(* IEC 61131-3 sources: Industry-PLC-LLM/data/PLCBEAD_repo/PLCBEAD_PLCEmbed-main/PLC-BEAD/Source/GEB/sample_project/oscat/Network (part 2) *)

(* ---- NET_VAR_BOOL8.ST ---- *)
TYPE

	oscat_NW_BUF_LONG  : ARRAY [0..4095] OF BYTE;

	oscat_NETWORK_BUFFER :
	STRUCT
		SIZE   : UINT;
		BUFFER : oscat_NW_BUF_LONG;
	END_STRUCT;

END_TYPE

TYPE oscat_NET_VAR_DATA :
	STRUCT
		CYCLE : UDINT;
		STATE : BYTE;
		INDEX : INT;
		ID_MAX : USINT;
		ERROR_ID : BYTE;
		BUF_SIZE : UINT;
		S_BUF : oscat_NETWORK_BUFFER;
		R_BUF : oscat_NETWORK_BUFFER;
	END_STRUCT;
END_TYPE

FUNCTION BIT_OF_DWORD : BOOL
  VAR_INPUT
    IN : DWORD;
    N : INT;
  END_VAR

  BIT_OF_DWORD := (SHR(IN,N) AND 16#00000001) > 0;
END_FUNCTION

FUNCTION_BLOCK BYTE_TO_BITS_Block
	VAR_INPUT
		IN :	BYTE;
	END_VAR

	VAR_OUTPUT
		B0 :	BOOL;
		B1 :	BOOL;
		B2 :	BOOL;
		B3 :	BOOL;
		B4 :	BOOL;
		B5 :	BOOL;
		B6 :	BOOL;
		B7 :	BOOL;
	END_VAR

	B0 := BIT_OF_DWORD(BYTE_TO_DWORD(IN),0); (* IN.X0 *)
	B1 := BIT_OF_DWORD(BYTE_TO_DWORD(IN),1); (* IN.X1 *)
	B2 := BIT_OF_DWORD(BYTE_TO_DWORD(IN),2); (* IN.X2 *)
	B3 := BIT_OF_DWORD(BYTE_TO_DWORD(IN),3); (* IN.X3 *)
	B4 := BIT_OF_DWORD(BYTE_TO_DWORD(IN),4); (* IN.X4 *)
	B5 := BIT_OF_DWORD(BYTE_TO_DWORD(IN),5); (* IN.X5 *)
	B6 := BIT_OF_DWORD(BYTE_TO_DWORD(IN),6); (* IN.X6 *)
	B7 := BIT_OF_DWORD(BYTE_TO_DWORD(IN),7); (* IN.X7 *)
END_FUNCTION_BLOCK

FUNCTION BYTE_OF_BIT:BYTE
	VAR_INPUT
		B0 :	BOOL;
		B1 :	BOOL;
		B2 :	BOOL;
		B3 :	BOOL;
		B4 :	BOOL;
		B5 :	BOOL;
		B6 :	BOOL;
		B7 :	BOOL;
	END_VAR
	Byte_of_bit := SHL(SHL(SHL(SHL(SHL(SHL(SHL(BOOL_TO_BYTE(B7),1) OR BOOL_TO_BYTE(B6),1)
	OR BOOL_TO_BYTE(B5),1) OR BOOL_TO_BYTE(B4),1) OR BOOL_TO_BYTE(B3),1) OR BOOL_TO_BYTE(B2),1)
	OR BOOL_TO_BYTE(B1),1) OR BOOL_TO_BYTE(B0);
END_FUNCTION

FUNCTION_BLOCK NET_VAR_BOOL8_Block

	VAR_INPUT
		IN1 :	BOOL;
		IN2 :	BOOL;
		IN3 :	BOOL;
		IN4 :	BOOL;
		IN5 :	BOOL;
		IN6 :	BOOL;
		IN7 :	BOOL;
		IN8 :	BOOL;
	END_VAR

	VAR_OUTPUT
		OUT1 :	BOOL;
		OUT2 :	BOOL;
		OUT3 :	BOOL;
		OUT4 :	BOOL;
		OUT5 :	BOOL;
		OUT6 :	BOOL;
		OUT7 :	BOOL;
		OUT8 :	BOOL;
		ID :	BYTE;
	END_VAR

	VAR_IN_OUT
		X :	oscat_NET_VAR_DATA;
	END_VAR

	VAR
		init :	BOOL;
		index :	INT;
		indeX2 :	INT;
		_BYTE_TO_BITS :	BYTE_TO_BITS_Block;
	END_VAR

	IF NOT init THEN
		init := TRUE;
		X.ID_MAX := X.ID_MAX + USINT#1;
		ID := USINT_TO_BYTE(X.ID_MAX);
	END_IF;

	IF X.STATE > BYTE#0 AND X.ERROR_ID = BYTE#0 THEN
		index := X.index;
		IF INT_TO_UINT(index + 3) > X.BUF_SIZE THEN
			X.ERROR_ID := ID;
		ELSE
			IF X.STATE = BYTE#1 THEN
				X.S_BUF.BUFFER[index] := ID;
				index := index + 1;
				X.S_BUF.BUFFER[index] := BYTE#4;
				index := index + 1;
				X.S_BUF.BUFFER[index] := BYTE_OF_BIT(IN1,IN2,IN3,IN4,IN5,IN6,IN7,IN8);
				index := index + 1;

			ELSIF X.STATE = BYTE#2 THEN
				indeX2 := index + 1;
				IF X.R_BUF.BUFFER[index] <> ID OR X.R_BUF.BUFFER[indeX2] <> BYTE#4 THEN
					X.ERROR_ID := ID;
				ELSE
					index := index + 2;
					_BYTE_TO_BITS(IN:=X.R_BUF.BUFFER[index]);
					OUT1 := _BYTE_TO_BITS.B0;
					OUT2 := _BYTE_TO_BITS.B1;
					OUT3 := _BYTE_TO_BITS.B2;
					OUT4 := _BYTE_TO_BITS.B3;
					OUT5 := _BYTE_TO_BITS.B4;
					OUT6 := _BYTE_TO_BITS.B5;
					OUT7 := _BYTE_TO_BITS.B6;
					OUT8 := _BYTE_TO_BITS.B7;
					index := index + 1;
				END_IF;
			END_IF;
			X.index := index;
		END_IF;
	END_IF;

END_FUNCTION_BLOCK

PROGRAM program0
	VAR
		IN1 :	BOOL;
		IN2 :	BOOL;
		IN3 :	BOOL;
		IN4 :	BOOL;
		IN5 :	BOOL;
		IN6 :	BOOL;
		IN7 :	BOOL;
		IN8 :	BOOL;
		OUT1 :	BOOL;
		OUT2 :	BOOL;
		OUT3 :	BOOL;
		OUT4 :	BOOL;
		OUT5 :	BOOL;
		OUT6 :	BOOL;
		OUT7 :	BOOL;
		OUT8 :	BOOL;
		ID :	BYTE;
		X :	oscat_NET_VAR_DATA;

		func_block : NET_VAR_BOOL8_Block;
	END_VAR
	func_block.IN1 := IN1;
	func_block.IN2 := IN2;
	func_block.IN3 := IN3;
	func_block.IN4 := IN4;
	func_block.IN5 := IN5;
	func_block.IN6 := IN6;
	func_block.IN7 := IN7;
	func_block.IN8 := IN8;
	func_block.X := X;

	func_block();
  	OUT1  := func_block.OUT1;
	OUT2  := func_block.OUT2;
	OUT3  := func_block.OUT3;
	OUT4  := func_block.OUT4;
	OUT5  := func_block.OUT5;
	OUT6  := func_block.OUT6;
	OUT7  := func_block.OUT7;
	OUT8  := func_block.OUT8;
	ID  := func_block.ID;
	X  := func_block.X;
END_PROGRAM

CONFIGURATION Config0
	RESOURCE ReS0 ON PLC
		TASK task0(INTERVAL := T#20ms,PRIORITY := 0);
		PROGRAM instance0 WITH task0 : program0;
	END_RESOURCE
END_CONFIGURATION

(* ---- NET_VAR_BUFFER.ST ---- *)
TYPE
	oscat_aB1_64 : ARRAY[1..64] OF BYTE;
END_TYPE

TYPE

	oscat_NW_BUF_LONG  : ARRAY [0..4095] OF BYTE;

	oscat_NETWORK_BUFFER :
	STRUCT
		SIZE   : UINT;
		BUFFER : oscat_NW_BUF_LONG;
	END_STRUCT;

END_TYPE

TYPE oscat_NET_VAR_DATA :
	STRUCT
		CYCLE : UDINT;
		STATE : BYTE;
		INDEX : INT;
		ID_MAX : USINT;
		ERROR_ID : BYTE;
		BUF_SIZE : UINT;
		S_BUF : oscat_NETWORK_BUFFER;
		R_BUF : oscat_NETWORK_BUFFER;
	END_STRUCT;
END_TYPE

FUNCTION_BLOCK NET_VAR_BUFFER_Block

	VAR_OUTPUT
		ID :	BYTE;
	END_VAR

	VAR_IN_OUT
		BUF_IN :	oscat_aB1_64;
		BUF_OUT :	oscat_aB1_64;
		X :	oscat_NET_VAR_DATA;
	END_VAR

	VAR
		SIZE :	INT;
		init :	BOOL;
		index :	INT;
		indeX2 :	INT;
	END_VAR

	IF NOT init THEN
		init := TRUE;
		X.ID_MAX := X.ID_MAX + USINT#1;
		ID := USINT_TO_BYTE(X.ID_MAX);
	END_IF;

	IF X.STATE > BYTE#0 AND X.ERROR_ID = BYTE#0 THEN
		index := X.index;
		IF X.STATE = BYTE#1 THEN
			SIZE := 64;
			IF INT_TO_UINT(index + 3 + SIZE) > X.BUF_SIZE THEN
				X.ERROR_ID := ID;
			ELSE
				X.S_BUF.BUFFER[index] := ID;
				index := index + 1;
				X.S_BUF.BUFFER[index] := BYTE#20;
				index := index + 1;
				X.S_BUF.BUFFER[index] := INT_TO_BYTE(SIZE);
				index := index + 1;
				FOR indeX2 := 1 TO SIZE DO
					X.S_BUF.BUFFER[index] := BUF_IN[indeX2];
					index := index + 1;
				END_FOR;
			END_IF;
		ELSIF X.STATE = BYTE#2 THEN
			indeX2 := index + 1;
			IF X.R_BUF.BUFFER[index] <> ID OR X.R_BUF.BUFFER[indeX2] <> BYTE#20 THEN
				X.ERROR_ID := ID;
			ELSE
				index := index + 2;
				SIZE := BYTE_TO_INT(X.R_BUF.BUFFER[index]);
				index := index + 1;
				FOR indeX2 := 1 TO SIZE DO
					BUF_OUT[indeX2] := X.R_BUF.BUFFER[index];
					index := index + 1;
				END_FOR;
			END_IF;
		END_IF;
		X.index := index;
	END_IF;

END_FUNCTION_BLOCK

PROGRAM program0
	VAR
		BUF_IN :	oscat_aB1_64;
		BUF_OUT :	oscat_aB1_64;
		X :	oscat_NET_VAR_DATA;
		ID :	BYTE;

		func_block : NET_VAR_BUFFER_Block;
	END_VAR
	func_block.BUF_IN := BUF_IN;
	func_block.BUF_OUT := BUF_OUT;
	func_block.X := X;

	func_block();
  	BUF_IN  := func_block.BUF_IN;
	BUF_OUT  := func_block.BUF_OUT;
	X  := func_block.X;
	ID  := func_block.ID;

END_PROGRAM

CONFIGURATION Config0
	RESOURCE ReS0 ON PLC
		TASK task0(INTERVAL := T#20ms,PRIORITY := 0);
		PROGRAM instance0 WITH task0 : program0;
	END_RESOURCE
END_CONFIGURATION

(* ---- NET_VAR_DWORD8.ST ---- *)
TYPE
	oscat_nv_dw : ARRAY[1..8] OF DWORD;
END_TYPE

TYPE

	oscat_NW_BUF_LONG  : ARRAY [0..4095] OF BYTE;

	oscat_NETWORK_BUFFER :
	STRUCT
		SIZE   : UINT;
		BUFFER : oscat_NW_BUF_LONG;
	END_STRUCT;

END_TYPE

TYPE oscat_NET_VAR_DATA :
	STRUCT
		CYCLE : UDINT;
		STATE : BYTE;
		INDEX : INT;
		ID_MAX : USINT;
		ERROR_ID : BYTE;
		BUF_SIZE : UINT;
		S_BUF : oscat_NETWORK_BUFFER;
		R_BUF : oscat_NETWORK_BUFFER;
	END_STRUCT;
END_TYPE

FUNCTION_BLOCK NET_VAR_DWORD8_Block

	VAR_INPUT
		IN1 :	DWORD;
		IN2 :	DWORD;
		IN3 :	DWORD;
		IN4 :	DWORD;
		IN5 :	DWORD;
		IN6 :	DWORD;
		IN7 :	DWORD;
		IN8 :	DWORD;
	END_VAR

	VAR_OUTPUT
		OUT1 :	DWORD;
		OUT2 :	DWORD;
		OUT3 :	DWORD;
		OUT4 :	DWORD;
		OUT5 :	DWORD;
		OUT6 :	DWORD;
		OUT7 :	DWORD;
		OUT8 :	DWORD;
		ID :	BYTE;
	END_VAR

	VAR_IN_OUT
		X :	oscat_NET_VAR_DATA;
	END_VAR

	VAR
		init :	BOOL;
		i :	INT;
		i2 :	INT;
		index :	INT;
		indeX2 :	INT;
		ra :	oscat_nv_dw;
	END_VAR

	IF NOT init THEN
		init := TRUE;
		X.ID_MAX := X.ID_MAX + USINT#1;
		ID := USINT_TO_BYTE(X.ID_MAX);
	END_IF;

	IF X.STATE > BYTE#0 AND X.ERROR_ID = BYTE#0 THEN
		index := X.index;
		IF INT_TO_UINT(index + 34) > X.BUF_SIZE THEN
			X.ERROR_ID := ID;
		ELSE
			IF X.STATE = BYTE#1 THEN
				ra[1] := IN1;
				ra[2] := IN2;
				ra[3] := IN3;
				ra[4] := IN4;
				ra[5] := IN5;
				ra[6] := IN6;
				ra[7] := IN7;
				ra[8] := IN8;
				X.S_BUF.BUFFER[index] := ID;
				index := index + 1;
				X.S_BUF.BUFFER[index] := BYTE#13;
				index := index + 1;
				FOR i2 := 1 TO 8 DO
					FOR i := 1 TO 4 DO
						X.S_BUF.BUFFER[index] := DWORD_TO_BYTE(ra[i2]);
						ra[i2] := ROR(ra[i2],8);
						index := index + 1;
					END_FOR;
				END_FOR;

			ELSIF X.STATE = BYTE#2 THEN
				indeX2 := index + 1;
				IF X.R_BUF.BUFFER[index] <> ID OR X.R_BUF.BUFFER[indeX2] <> BYTE#13 THEN
					X.ERROR_ID := ID;
				ELSE
					index := index + 2;
					FOR i2 := 1 TO 8 DO
						ra[i2] := DWORD#0;
						FOR i := 1 TO 4 DO
							ra[i2] := ra[i2] OR BYTE_TO_DWORD(X.R_BUF.BUFFER[index]);
							ra[i2] := ROR(ra[i2],8);
							index := index + 1;
						END_FOR;
					END_FOR;
					OUT1 := ra[1];
					OUT2 := ra[2];
					OUT3 := ra[3];
					OUT4 := ra[4];
					OUT5 := ra[5];
					OUT6 := ra[6];
					OUT7 := ra[7];
					OUT8 := ra[8];
				END_IF;
			END_IF;
			X.index := index;
		END_IF;
	END_IF;

END_FUNCTION_BLOCK

PROGRAM program0
	VAR
		IN1 :	DWORD;
		IN2 :	DWORD;
		IN3 :	DWORD;
		IN4 :	DWORD;
		IN5 :	DWORD;
		IN6 :	DWORD;
		IN7 :	DWORD;
		IN8 :	DWORD;
		OUT1 :	DWORD;
		OUT2 :	DWORD;
		OUT3 :	DWORD;
		OUT4 :	DWORD;
		OUT5 :	DWORD;
		OUT6 :	DWORD;
		OUT7 :	DWORD;
		OUT8 :	DWORD;
		ID :	BYTE;
		X :	oscat_NET_VAR_DATA;

		func_block : NET_VAR_DWORD8_Block;
	END_VAR
	func_block.IN1 := IN1;
	func_block.IN2 := IN2;
	func_block.IN3 := IN3;
	func_block.IN4 := IN4;
	func_block.IN5 := IN5;
	func_block.IN6 := IN6;
	func_block.IN7 := IN7;
	func_block.IN8 := IN8;
	func_block.X := X;

	func_block();
  	OUT1  := func_block.OUT1;
	OUT2  := func_block.OUT2;
	OUT3  := func_block.OUT3;
	OUT4  := func_block.OUT4;
	OUT5  := func_block.OUT5;
	OUT6  := func_block.OUT6;
	OUT7  := func_block.OUT7;
	OUT8  := func_block.OUT8;
	ID  := func_block.ID;
	X  := func_block.X;
END_PROGRAM

CONFIGURATION Config0
	RESOURCE ReS0 ON PLC
		TASK task0(INTERVAL := T#20ms,PRIORITY := 0);
		PROGRAM instance0 WITH task0 : program0;
	END_RESOURCE
END_CONFIGURATION

(* ---- SHA1_STREAM.ST ---- *)
TYPE
  oscat_aB0_19	: ARRAY [0..19]	OF BYTE;
  oscat_aB0_63	: ARRAY [0..63]	OF BYTE;
  oscat_aDW0_4	: ARRAY [0..4] 	OF DWORD;
  oscat_sDW0_79	: ARRAY [0..79] OF DWORD;

END_TYPE

FUNCTION DWORD_OF_BYTE:DWORD
	VAR_INPUT
		B3 :	BYTE;
		B2 :	BYTE;
		B1 :	BYTE;
		B0 :	BYTE;
	END_VAR

	DWORD_OF_BYTE := SHL(SHL(SHL(BYTE_TO_DWORD(B3),8) OR BYTE_TO_DWORD(B2),8) OR BYTE_TO_DWORD(B1),8) OR BYTE_TO_DWORD(B0);

END_FUNCTION

FUNCTION_BLOCK SHA1_STREAM_Block

	VAR_IN_OUT
		MODE :	INT;
		BUF :	oscat_aB0_63;
		SHA1 :	oscat_aB0_19;
		SIZE :	UDINT;
	END_VAR

	VAR_OUTPUT
		POS :	UDINT;
	END_VAR

	VAR
		hash :	oscat_aDW0_4;
		end :	UDINT;
		block :	UDINT;
		pad_1 :	BOOL;
		w :	oscat_sDW0_79;
		n :	INT;
		n1 :	INT;
		n2 :	INT;
		n3 :	INT;
		n4 :	INT;
		a :	DWORD;
		b :	DWORD;
		c :	DWORD;
		d :	DWORD;
		e :	DWORD;
		f :	DWORD;
		k :	DWORD;
		x :	DWORD;
	END_VAR

	CASE MODE OF

	1:
		hash[0] := DWORD#16#67452301;
		hash[1] := DWORD#16#EFCDAB89;
		hash[2] := DWORD#16#98BADCFE;
		hash[3] := DWORD#16#10325476;
		hash[4] := DWORD#16#C3D2E1F0;

		FOR n := 16 TO 79 DO
			w[n] := DWORD#0;
		END_FOR;

		block := DWORD_TO_UDINT(SHR(UDINT_TO_DWORD(SIZE),6)) + BOOL_TO_UDINT((UDINT_TO_BYTE(SIZE) AND BYTE#16#3F) > BYTE#55);

		pad_1 := FALSE;
		POS := UDINT#0;
		End := SIZE;
		SIZE := MIN(UDINT#64,End);
		MODE := 2;

	2:	FOR n := UDINT_TO_INT(SIZE) TO 63 DO
			BUF[n] := BYTE#0;
		END_FOR;

		IF SIZE < UDINT#64 AND NOT pad_1 THEN
			BUF[SIZE] := BYTE#2#1000_0000;
			pad_1 := TRUE;
		END_IF;

		POS := POS + SIZE;
		SIZE := MIN(UDINT#64,End - POS);

		n := 0;
		FOR n4 := 0 TO 15 DO
			n1 := n + 1;
			n2 := n + 2;
			n3 := n + 3;
			w[n4] := DWORD_OF_BYTE(BUF[n],BUF[n1],BUF[n2],BUF[n3]);
			n := n + 4;
		END_FOR;

		IF block = UDINT#0 THEN
			w[15] := SHL(UDINT_TO_DWORD(End),3);
			MODE := 3;
		ELSE
			block := block - UDINT#1;
		END_IF;

		FOR n := 16 TO 79 DO
			n1 := n - 3;
			n2 := n - 8;
			n3 := n - 14;
			n4 := n - 16;
			w[n] := ROL(w[n1] XOR w[n2] XOR w[n3] XOR w[n4],1);
		END_FOR;

		a := hash[0];
		b := hash[1];
		c := hash[2];
		d := hash[3];
		e := hash[4];

		FOR n := 0 TO 79 DO
			IF n <= 19 THEN
				f := (b AND c) OR (NOT(b) AND d);
				k := DWORD#16#5A827999;
			ELSIF n <= 39 THEN
				f := b XOR c XOR d;
				k := DWORD#16#6ED9EBA1;
			ELSIF n <= 59 THEN
				f := (b AND c) OR (b AND d) OR (c AND d);
				k := DWORD#16#8F1BBCDC;
			ELSE
				f := b XOR c XOR d;
				k := DWORD#16#CA62C1D6;
			END_IF;

			x := UDINT_TO_DWORD(DWORD_TO_UDINT(ROL(a,5)) + DWORD_TO_UDINT(f) + DWORD_TO_UDINT(e) + DWORD_TO_UDINT(k) + DWORD_TO_UDINT(w[n]));
			e := d;
			d := c;
			c := ROL(b,30);
			b := a;
			a := x;
		END_FOR;

		hash[0] := UDINT_TO_DWORD(DWORD_TO_UDINT(hash[0]) + DWORD_TO_UDINT(a));
		hash[1] := UDINT_TO_DWORD(DWORD_TO_UDINT(hash[1]) + DWORD_TO_UDINT(b));
		hash[2] := UDINT_TO_DWORD(DWORD_TO_UDINT(hash[2]) + DWORD_TO_UDINT(c));
		hash[3] := UDINT_TO_DWORD(DWORD_TO_UDINT(hash[3]) + DWORD_TO_UDINT(d));
		hash[4] := UDINT_TO_DWORD(DWORD_TO_UDINT(hash[4]) + DWORD_TO_UDINT(e));

	END_CASE;

	IF MODE = 3 THEN
		n2 := 0;
		FOR n := 0 TO 4 DO
			FOR n1 := 0 TO 3 DO
				hash[n] := ROL(hash[n],8);
				SHA1[n2] := DWORD_TO_BYTE(hash[n]);
				n2 := n2 + 1;
			END_FOR;
		END_FOR;
	END_IF;

END_FUNCTION_BLOCK

PROGRAM program0
	VAR
		MODE :	INT;
		BUF :	oscat_aB0_63;
		SHA1 :	oscat_aB0_19;
		SIZE :	UDINT;
		POS :	UDINT;

		func_block : SHA1_STREAM_Block;
	END_VAR
	func_block.MODE := MODE;
	func_block.BUF := BUF;
	func_block.SHA1 := SHA1;
	func_block.SIZE := SIZE;

	func_block();
  	MODE  := func_block.MODE;
	BUF  := func_block.BUF;
	SHA1  := func_block.SHA1;
	SIZE  := func_block.SIZE;
	POS  := func_block.POS;
END_PROGRAM

CONFIGURATION Config0
	RESOURCE ReS0 ON PLC
		TASK task0(INTERVAL := T#20ms,PRIORITY := 0);
		PROGRAM instance0 WITH task0 : program0;
	END_RESOURCE
END_CONFIGURATION

(* ---- SNTP_CLIENT.ST ---- *)
TYPE
  oscat_IP_FIFO128_DATA  : ARRAY [1..128] OF BYTE;
  oscat_Mailbox  : ARRAY [1..16] OF BYTE;

  oscat_IP_FIFO_DATA :
  STRUCT
    X       : oscat_IP_FIFO128_DATA; (* IP_ID FIFO Speicher          *)
    Y       : oscat_IP_FIFO128_DATA; (* IP_ID Z�hler                 *)
    ID      : BYTE;                  (* h�chste vergabene id         *)
    MAX_ID  : BYTE;                  (* maximal Anmeldungen pro ID   *)
      INIT    : BOOL;                  (* Initialisierung durchgef�hrt *)
    EMPTY   : BOOL;                  (* FIFO leer                    *)
    FULL    : BOOL;                  (* FIFO voll                    *)
    TOP     : INT;                   (* maximale anzahl IN FIFO      *)
    NW      : INT;                   (* Schreibzeiger                *)
    NR      : INT;                   (* Lesezeiger                   *)
  END_STRUCT;

  oscat_IP_C:
  STRUCT
    C_MODE:			BYTE;          		(*W Mode: TCP/UCP AKTIV/PASSIV                               *)
    C_PORT:         WORD;          		(*W Portnummer                                               *)
    C_IP:           DWORD;         		(*W IP-ADRESSe gepackt wwxxyyzz = www.xxx.yyy.zzz            *)
    C_STATE:        BYTE;          		(*R VerbindungsSTATUS ON/OFF + Flanke ON/OFF                 *)
    C_ENABLE:       BOOL;          		(*W Freigabe f�r Connect                                     *)
    R_OBSERVE:      BOOL;          		(*W Empfang ueberwachen                                      *)
    TIME_RESET:     BOOL;          		(*W Alle Timer ruecksetzen                                   *)
    ERROR:          DWORD;         		(*R vvwwxxyy (vv = CON_ERROR, ww = SEN_ERROR, xx = REC_ERROR *)
    FIFO:           oscat_IP_FIFO_DATA; (*I IP FIFO Struktur                                         *)
    MAILBOX:		oscat_Mailbox;		(*I Mailbox: Datenbereich f�r Bausteindatenaustausch         *)
  END_STRUCT;
END_TYPE

TYPE

  oscat_NW_BUF_LONG  : ARRAY [0..4095] OF BYTE;

  oscat_NETWORK_BUFFER :
  STRUCT
    SIZE   : UINT;
    BUFFER : oscat_NW_BUF_LONG;
  END_STRUCT;

END_TYPE

FUNCTION _BYTE_TO_INT:INT
	VAR_INPUT
		IN :	BYTE;
	END_VAR

	_BYTE_TO_INT := USINT_TO_INT(BYTE_TO_USINT(IN));
END_FUNCTION

FUNCTION_BLOCK IP_FIFO_Block

  VAR_IN_OUT
    FIFO :	oscat_IP_FIFO_DATA;
    ID :	BYTE;
    STATE :	BYTE;
  END_VAR

  VAR
    tmp :	INT;
  END_VAR

  IF NOT FIFO.INIT THEN
    FIFO.INIT		:= TRUE;
    FIFO.NW		:= 1;
    FIFO.NR		:= 1;
    FIFO.EMPTY	:= TRUE;
    FIFO.FULL		:= FALSE;
    FIFO.TOP		:= 128;
    FIFO.MAX_ID	:= BYTE#1;
  END_IF;

  IF ID = BYTE#00 THEN
    IF FIFO.ID < INT_TO_BYTE(FIFO.TOP) THEN
      ID := USINT_TO_BYTE(BYTE_TO_USINT(FIFO.ID) + USINT#1);
      FIFO.ID := ID ;

    ELSIF STATE < BYTE#200 THEN
      STATE := BYTE#255;
    RETURN;
    END_IF;
  END_IF;

  IF STATE = BYTE#1 AND NOT FIFO.FULL THEN
    tmp := _BYTE_TO_INT(ID);
    IF FIFO.Y[tmp] < FIFO.MAX_ID THEN
      FIFO.Y[tmp] := USINT_TO_BYTE(BYTE_TO_USINT(FIFO.Y[tmp]) + USINT#1);
      tmp := FIFO.NW;
      FIFO.X[tmp] := ID;
      IF FIFO.NW = FIFO.TOP THEN FIFO.NW := 1; ELSE FIFO.NW := FIFO.NW + 1; END_IF;
      FIFO.FULL := FIFO.NW = FIFO.NR;
    FIFO.EMPTY := FALSE;
      STATE := BYTE#2;
    END_IF;
  END_IF;

  IF STATE = BYTE#2 AND NOT FIFO.EMPTY THEN
    tmp := FIFO.NR;
    IF ID = FIFO.X[tmp] THEN
      STATE := BYTE#3;
    END_IF;
  END_IF;

  IF STATE = BYTE#4 AND NOT FIFO.EMPTY THEN

    tmp := FIFO.NR;
    IF ID = FIFO.X[tmp] THEN
      tmp := _BYTE_TO_INT(ID);
      FIFO.Y[tmp] := USINT_TO_BYTE(BYTE_TO_USINT(FIFO.Y[tmp]) - USINT#1);

      IF FIFO.NR = FIFO.TOP THEN FIFO.NR := 1; ELSE FIFO.NR := FIFO.NR + 1; END_IF;
      FIFO.EMPTY := FIFO.NR = FIFO.NW;
    FIFO.FULL := FALSE;
    END_IF;
    STATE := BYTE#5;
  END_IF;

END_FUNCTION_BLOCK

FUNCTION_BLOCK T_PLC_MS_block

	VAR_OUTPUT
		T_PLC_MS :	UDINT;
	END_VAR

	VAR
		PLC_TICKS_PER_SEC :	INT;
		PLC_SYS_TICK_CNT :	DINT;
	END_VAR

	VAR
		debug :	BOOL;(*Debug-Mode ON / OFF*)
		N :	INT;(*Debug-Faktor*)
		Offset :	UDINT;(*Debug-Offset*)
		temp :	DWORD := DWORD#1;(*Debug-Offset*)
		MODE :	BOOL;(*modus*)
		faktor :	UDINT;(*Systemtakt-Faktor*)
		init :	BOOL;
		v_plc_ticks_per_sec :	UDINT;
		base :	UDINT := UDINT#1000;
	END_VAR

	IF init = FALSE THEN
		v_plc_ticks_per_sec := INT_TO_UDINT(PLC_TICKS_PER_SEC);
		IF v_plc_ticks_per_sec = UDINT#1024 THEN
			faktor := UDINT#1;
			MODE := FALSE;
		ELSIF v_plc_ticks_per_sec > UDINT#0 THEN
			IF v_plc_ticks_per_sec <= base THEN
				faktor := base / v_plc_ticks_per_sec;
				MODE := FALSE;
			ELSE
				faktor := v_plc_ticks_per_sec / base;
				MODE := TRUE;
			END_IF;
		ELSE
			faktor := UDINT#1;
		END_IF;
		init := TRUE;
	END_IF;

	IF MODE THEN
		T_PLC_MS := DINT_TO_UDINT(PLC_SYS_TICK_CNT) / faktor;
	ELSE
		T_PLC_MS := DINT_TO_UDINT(PLC_SYS_TICK_CNT) * faktor;
	END_IF;

	IF debug THEN
		T_PLC_MS := (DWORD_TO_UDINT(SHL(UDINT_TO_DWORD(T_PLC_MS),N) OR SHL(temp,N)) - UDINT#1) + Offset;
	END_IF;

END_FUNCTION_BLOCK

FUNCTION DWORD_OF_BYTE:DWORD
	VAR_INPUT
		B3 :	BYTE;
		B2 :	BYTE;
		B1 :	BYTE;
		B0 :	BYTE;
	END_VAR

	DWORD_OF_BYTE := SHL(SHL(SHL(BYTE_TO_DWORD(B3),8) OR BYTE_TO_DWORD(B2),8) OR BYTE_TO_DWORD(B1),8) OR BYTE_TO_DWORD(B0);

END_FUNCTION

FUNCTION _WORD_TO_DINT:DINT
	VAR_INPUT
		IN :	WORD;
	END_VAR
	_WORD_TO_DINT := UINT_TO_DINT(WORD_TO_UINT(IN));
END_FUNCTION

FUNCTION WORD_OF_BYTE:WORD
	VAR_INPUT
		B1 :	BYTE;
		B0 :	BYTE;
	END_VAR
	WORD_OF_BYTE := SHL(BYTE_TO_WORD(B1),8) OR BYTE_TO_WORD(B0);
END_FUNCTION

FUNCTION _INT_TO_UDINT:UDINT
	VAR_INPUT
		IN :	INT;
	END_VAR

	_INT_TO_UDINT := DINT_TO_UDINT(INT_TO_DINT(IN));
END_FUNCTION

FUNCTION_BLOCK SNTP_CLIENT_Block

  VAR_IN_OUT
    IP_C :	oscat_IP_C;
    S_BUF :	oscat_NETWORK_BUFFER;
    R_BUF :	oscat_NETWORK_BUFFER;
  END_VAR

  VAR_INPUT
    IP4 :	DWORD;
    ACTIVATE :	BOOL;
  END_VAR

  VAR_OUTPUT
    ERROR :	DWORD;
    DONE_P :	BOOL;
    UDT :	UDINT;
    XMS :	INT;
  END_VAR

  VAR
    IP_STATE :	BYTE;
    IP_ID :	BYTE;
    IP_FIFO :	IP_FIFO_Block;
    i :	INT;
    last :	UDINT;
    STATE :	INT;
    T_PLC_MS :	T_PLC_MS_block;
    TX :	UDINT;
    ACTIVATE_LAST :	BOOL;
    IP4_STORED :	DWORD;
  END_VAR

  T_PLC_MS();
  TX := T_PLC_MS.T_PLC_MS;

  CASE STATE OF
  00:
    DONE_P := FALSE;
    IF ACTIVATE AND NOT ACTIVATE_LAST THEN
      IP4_STORED := IP4;
      STATE := 10;
      ERROR := DWORD#0;
      IP_STATE := BYTE#1;
    END_IF;

  10:
    IF IP_STATE = BYTE#3 THEN

      S_BUF.BUFFER[00] := BYTE#16#1B;
      FOR i := 1 TO 47 DO
        S_BUF.BUFFER[i] := BYTE#16#00;
      END_FOR;

      last := TX;
      STATE := 30;

      IP_C.C_PORT     := WORD#123;
      IP_C.C_IP       := IP4_STORED;
      IP_C.C_MODE     := BYTE#1;
      IP_C.C_ENABLE   := TRUE;
      IP_C.TIME_RESET := TRUE;
      IP_C.R_OBSERVE  := TRUE;
      S_BUF.SIZE      := UINT#48;
      R_BUF.SIZE      := UINT#0;
    END_IF;

  30:
    IF IP_C.ERROR <> DWORD#00 THEN
      ERROR := IP_C.ERROR;
    S_BUF.SIZE := UINT#0;
    R_BUF.SIZE := UINT#0;
      STATE := 0;
    ELSIF S_BUF.SIZE = UINT#0 AND R_BUF.SIZE >= UINT#48 THEN
      UDT := DWORD_TO_UDINT(DWORD_OF_BYTE(R_BUF.BUFFER[40],R_BUF.BUFFER[41],R_BUF.BUFFER[42],R_BUF.BUFFER[43]))- UDINT#2208988800;

      XMS := DWORD_TO_INT(SHR(DINT_TO_DWORD(_WORD_TO_DINT(WORD_OF_BYTE(R_BUF.BUFFER[44],R_BUF.BUFFER[45])) * DINT#1000),16));
      XMS := XMS + DWORD_TO_INT(SHR(UDINT_TO_DWORD(SUB_TIME(TX, last)),1));

      UDT := UDT + _INT_TO_UDINT(XMS / 1000);
      XMS := XMS MOD 1000;

      STATE := 0;
      DONE_P := TRUE;

    END_IF;

    IF STATE = 0 THEN
      IP_C.R_OBSERVE := FALSE;
      IP_STATE := BYTE#4;
    END_IF;

  END_CASE;

  ACTIVATE_LAST := ACTIVATE;

  IP_FIFO(FIFO:=IP_C.FIFO,STATE:=IP_STATE,ID:=IP_ID);
  IP_C.FIFO:=IP_FIFO.FIFO;
  IP_STATE := IP_FIFO.STATE;
  IP_ID:=IP_FIFO.ID;

END_FUNCTION_BLOCK

PROGRAM program0
	VAR
		IP_C :	oscat_IP_C;
    S_BUF :	oscat_NETWORK_BUFFER;
    R_BUF :	oscat_NETWORK_BUFFER;
    IP4 :	DWORD;
    ACTIVATE :	BOOL;
    ERROR :	DWORD;
    DONE_P :	BOOL;
    UDT :	UDINT;
    XMS :	INT;

		func_block : SNTP_CLIENT_Block;
	END_VAR
	func_block.IP_C := IP_C;
	func_block.S_BUF := S_BUF;
	func_block.R_BUF := R_BUF;
  func_block.IP4 := IP4;
	func_block.ACTIVATE := ACTIVATE;

	func_block();
  IP_C  := func_block.IP_C;
  S_BUF  := func_block.S_BUF;
  R_BUF  := func_block.R_BUF;
  ERROR  := func_block.ERROR;
  DONE_P  := func_block.DONE_P;
  UDT  := func_block.UDT;
  XMS  := func_block.XMS;
END_PROGRAM

CONFIGURATION Config0

	VAR_GLOBAL
		PLC_TICKS_PER_SEC :	INT;
		PLC_SYS_TICK_CNT :	DINT;
	END_VAR

  	RESOURCE ReS0 ON PLC
    	TASK task0(INTERVAL := T#20ms,PRIORITY := 0);
    	PROGRAM instance0 WITH task0 : program0;
  	END_RESOURCE

END_CONFIGURATION

(* ---- STRING_TO_URL.ST ---- *)
TYPE
  oscat_STRING250             : STRING;
  oscat_STRING32             : STRING;
  oscat_STRING80             : STRING;
  oscat_STRING160             : STRING;
  oscat_STRING40             : STRING;
  oscat_STRING10             : STRING;
  oscat_STRING20             : STRING;
END_TYPE

TYPE oscat_url :
    STRUCT
    PROTOCOL : oscat_STRING10;
    USER     : oscat_STRING32;
    PASSWORD : oscat_STRING32;
    DOMAIN   : oscat_STRING80;
    PORT     : WORD;
    PATH     : oscat_STRING80;
    QUERY    : oscat_STRING250;
    ANCHOR   : oscat_STRING40;
    HEADER   : oscat_STRING160;
    END_STRUCT;
END_TYPE

FUNCTION_BLOCK STRING_TO_URL_Block

	VAR_INPUT
		STR :	oscat_STRING250;
		DEFAULT_PROTOCOL :	oscat_STRING20 := 'http';
		DEFAULT_PATH :	oscat_STRING80 := '/';
	END_VAR

	VAR_OUTPUT
		STRING_TO_URL :	oscat_url;
	END_VAR

	VAR
		POS :	INT;
		POS2 :	INT;
		temp :	STRING;
		x :	oscat_STRING250;
	END_VAR

	IF EQ_STRING(STR,'') THEN
		RETURN;
	END_IF;

	POS := FIND(STR, '://');
	IF POS > 0 THEN
		STRING_TO_URL.PROTOCOL := LEFT(STR, POS - 1);
		x := RIGHT(STR, LEN(STR) - POS - 2);
	ELSE
		x := STR;
		STRING_TO_URL.PROTOCOL := DEFAULT_PROTOCOL;
	END_IF;

	POS := FIND(x, '@');
	IF POS > 0 THEN
		POS2 := FIND(x,':')+1;
		IF POS2 > 1 AND POS2 <= POS THEN
			STRING_TO_URL.USER := LEFT(x,POS2 - 2);
			STRING_TO_URL.PASSWORD := MID(x, POS - POS2, POS2);
		ELSE
			STRING_TO_URL.USER := LEFT(x, POS - 2);
			STRING_TO_URL.PASSWORD := '';
		END_IF;
		x := RIGHT(x, LEN(X) - POS);
	ELSE
		STRING_TO_URL.USER := '';
		STRING_TO_URL.PASSWORD := '';
	END_IF;

	POS := FIND(x, '#');
	IF POS > 0 THEN
		STRING_TO_URL.ANCHOR := RIGHT(x, LEN(X) - POS);
		x := LEFT(x, POS - 1);
	ELSE
		STRING_TO_URL.ANCHOR := '';
	END_IF;

	POS := FIND(x, '?');
	IF POS > 0 THEN
		STRING_TO_URL.QUERY := RIGHT(x, LEN(X) - POS);
		x := LEFT(x, POS - 1);
	ELSE
		STRING_TO_URL.QUERY := '';
	END_IF;

	POS := FIND(x, '/');
	IF POS > 0 THEN
		STRING_TO_URL.PATH := RIGHT(x, LEN(X) - POS + 1);
		x := LEFT(x, POS - 1);
	ELSE
		STRING_TO_URL.PATH := DEFAULT_PATH;
	END_IF;

	POS := FIND(x, ':');
	IF POS > 0 THEN
		temp := RIGHT(x, LEN(X) - POS);
		STRING_TO_URL.PORT := STRING_TO_WORD(temp);
		STRING_TO_URL.DOMAIN := LEFT(x, POS - 1);
	ELSE
		STRING_TO_URL.PORT := WORD#0;
		STRING_TO_URL.DOMAIN := x;
	END_IF;

END_FUNCTION_BLOCK

PROGRAM program0
	VAR
		STR :	oscat_STRING250;
		DEFAULT_PROTOCOL :	oscat_STRING20 := 'http';
		DEFAULT_PATH :	oscat_STRING80 := '/';
		STRING_TO_URL :	oscat_url;

		func_block : STRING_TO_URL_Block;
	END_VAR
	func_block.STR := STR;
	func_block.DEFAULT_PROTOCOL := DEFAULT_PROTOCOL;
	func_block.DEFAULT_PATH := DEFAULT_PATH;

	func_block();
  	STRING_TO_URL  := func_block.STRING_TO_URL;
END_PROGRAM

CONFIGURATION Config0
	RESOURCE ReS0 ON PLC
		TASK task0(INTERVAL := T#20ms,PRIORITY := 0);
		PROGRAM instance0 WITH task0 : program0;
	END_RESOURCE
END_CONFIGURATION

(* ---- TN_RECEIVE.ST ---- *)
TYPE
  bya_TN_CHAR:       	ARRAY [0..1919] OF BYTE;
  bya_TN_BACKUP:     	ARRAY [0..1919] OF BYTE;
  bya_TN_COLOR:      	ARRAY [0..1919] OF BYTE;
  bya_TN_Line_Update:	ARRAY [0..23]   OF BOOL;

  us_TN_SCREEN :
  STRUCT
		bya_CHAR:			bya_TN_CHAR;
		bya_COLOR:			bya_TN_COLOR;
		bya_BACKUP:			bya_TN_BACKUP;
		bya_Line_Update:	bya_TN_Line_Update;

		by_Input_Exten_Code:    BYTE;
		by_Input_ASCII_Code:    BYTE;
		bo_Input_ASCII_IsNum:   BOOL;
		in_Page_Number:        	INT;
		in_Cursor_X:           	INT;
		in_Cursor_Y:           	INT;
		in_EOS_Offset:         	INT;
		by_Clear_Screen_Attr:  	BYTE;
		bo_Clear_Screen:       	BOOL;
		bo_Modal_Dialog:       	BOOL;
		bo_Menue_Bar_Dialog:   	BOOL;

  END_STRUCT;
END_TYPE

TYPE
  oscat_NW_BUF_LONG  : ARRAY [0..4095] OF BYTE;

  oscat_NETWORK_BUFFER :
  STRUCT
    SIZE   : UINT;
    BUFFER : oscat_NW_BUF_LONG;
  END_STRUCT;
END_TYPE

FUNCTION ISC_NUM:BOOL

	VAR_INPUT
		IN :	BYTE;
	END_VAR

	ISC_NUM := IN > BYTE#47 AND IN < BYTE#58;

END_FUNCTION

FUNCTION_BLOCK TN_RECEIVE_Block

  VAR_IN_OUT
    R_BUF :	oscat_NETWORK_BUFFER;
    Xus_TN_SCREEN :	us_TN_SCREEN;
  END_VAR

  VAR
    REQ_SIZE :	UINT;
    REQ1 :	BYTE;
    REQ2 :	BYTE;
    REQ3 :	BYTE;
  END_VAR

  Xus_TN_SCREEN.by_Input_ASCII_Code := BYTE#00;
  Xus_TN_SCREEN.by_Input_Exten_Code := BYTE#00;

  IF R_BUF.SIZE > UINT#0 THEN
    REQ_SIZE := R_BUF.SIZE;
    REQ1 := R_BUF.BUFFER[0];
    REQ2 := R_BUF.BUFFER[1];
    REQ3 := R_BUF.BUFFER[2];

    IF REQ1 = BYTE#27 AND REQ_SIZE >= UINT#3 THEN
      IF REQ2 = BYTE#91 THEN
        IF (REQ3 >= BYTE#65 AND REQ3 <= BYTE#68) OR (REQ3 = BYTE#72) OR (REQ3 = BYTE#75) THEN
          Xus_TN_SCREEN.by_Input_Exten_Code := REQ3;
        END_IF;
      ELSIF REQ2 = BYTE#79 THEN
        IF REQ3 >= BYTE#80 AND REQ3 <= BYTE#83 THEN
          Xus_TN_SCREEN.by_Input_Exten_Code := REQ3;
        END_IF;
      END_IF;
    ELSIF REQ1 >= BYTE#32 AND REQ1 <= BYTE#126 THEN
    Xus_TN_SCREEN.by_Input_ASCII_Code := REQ1;
      Xus_TN_SCREEN.bo_Input_ASCII_IsNum := ISC_NUM(REQ1);
    ELSIF REQ1 = BYTE#8 OR REQ1 = BYTE#9 OR REQ1 = BYTE#13 OR REQ1 = BYTE#27 THEN
    Xus_TN_SCREEN.by_Input_Exten_Code := REQ1;
    END_IF;

    R_BUF.SIZE := UINT#00;
  END_IF;

END_FUNCTION_BLOCK

PROGRAM program0
	VAR
		R_BUF :	oscat_NETWORK_BUFFER;
    Xus_TN_SCREEN :	us_TN_SCREEN;

		func_block : TN_RECEIVE_Block;
	END_VAR
	func_block.R_BUF := R_BUF;
	func_block.Xus_TN_SCREEN := Xus_TN_SCREEN;

	func_block();
  R_BUF  := func_block.R_BUF;
	Xus_TN_SCREEN  := func_block.Xus_TN_SCREEN;
END_PROGRAM

CONFIGURATION Config0
	RESOURCE ReS0 ON PLC
		TASK task0(INTERVAL := T#20ms,PRIORITY := 0);
		PROGRAM instance0 WITH task0 : program0;
	END_RESOURCE
END_CONFIGURATION

(* ---- TN_SC_ADD_SHADOW.ST ---- *)
TYPE
  bya_TN_CHAR:       	ARRAY [0..1919] OF BYTE;
  bya_TN_BACKUP:     	ARRAY [0..1919] OF BYTE;
  bya_TN_COLOR:      	ARRAY [0..1919] OF BYTE;
  bya_TN_Line_Update:	ARRAY [0..23]   OF BOOL;

  us_TN_SCREEN :
  STRUCT
		bya_CHAR:			bya_TN_CHAR;
		bya_COLOR:			bya_TN_COLOR;
		bya_BACKUP:			bya_TN_BACKUP;
		bya_Line_Update:	bya_TN_Line_Update;

		by_Input_Exten_Code:    BYTE;
		by_Input_ASCII_Code:    BYTE;
		bo_Input_ASCII_IsNum:   BOOL;
		in_Page_Number:        	INT;
		in_Cursor_X:           	INT;
		in_Cursor_Y:           	INT;
		in_EOS_Offset:         	INT;
		by_Clear_Screen_Attr:  	BYTE;
		bo_Clear_Screen:       	BOOL;
		bo_Modal_Dialog:       	BOOL;
		bo_Menue_Bar_Dialog:   	BOOL;

  END_STRUCT;
END_TYPE

FUNCTION TN_SC_XY2_ERROR:BOOL

	VAR_INPUT
		X1 :	INT;
		Y1 :	INT;
		X2 :	INT;
		Y2 :	INT;
	END_VAR

	TN_SC_XY2_ERROR := Y1 < 0 OR X1 < 0 OR Y2 < 0 OR X2 < 0 OR Y1 > 23 OR X1 > 79 OR Y2 > 23 OR X2 > 79;

END_FUNCTION

FUNCTION TN_SC_SHADOW_ATTR:BYTE

	VAR_INPUT
		Iby_ATTR :	BYTE;
	END_VAR

	TN_SC_SHADOW_ATTR := ((Iby_ATTR AND BYTE#2#11110000) OR BYTE#2#00001000);

END_FUNCTION

FUNCTION_BLOCK TN_SC_ADD_SHADOW_Block

  VAR
    in_Offset :	INT;
    in_X :	INT;
    in_Y :	INT;
  END_VAR

  VAR_INPUT
    Iin_Y1 :	INT;
    Iin_X1 :	INT;
    Iin_Y2 :	INT;
    Iin_X2 :	INT;
    Iin_OPTION :	INT;
  END_VAR

  VAR_IN_OUT
    Xus_TN_SCREEN :	us_TN_SCREEN;
  END_VAR

  IF TN_SC_XY2_ERROR(Iin_X1,Iin_Y1,Iin_X2,Iin_Y2) THEN RETURN; END_IF;

  in_Offset := (Iin_Y1 * 80) + Iin_X2;

  IF Iin_OPTION = INT#00 THEN
    FOR in_Y := Iin_Y1 TO Iin_Y2 DO
      Xus_TN_SCREEN.bya_COLOR[in_Offset] := TN_SC_SHADOW_ATTR(Xus_TN_SCREEN.bya_COLOR[in_Offset]);
      in_Offset := in_Offset + 80;
      Xus_TN_SCREEN.bya_Line_Update[in_Y] := TRUE;
    END_FOR;
  ELSE
    FOR in_Y := Iin_Y1 TO Iin_Y2 DO
      Xus_TN_SCREEN.bya_COLOR[in_Offset] := BYTE#00;
      Xus_TN_SCREEN.bya_CHAR[in_Offset]  := BYTE#32;
      in_Offset := in_Offset + 80;
      Xus_TN_SCREEN.bya_Line_Update[in_Y] := TRUE;
    END_FOR;
  END_IF;

  in_Offset := (Iin_Y2 * 80) + Iin_X1;

  IF Iin_OPTION = INT#00 THEN
    FOR in_X  := Iin_X1 TO Iin_X2 DO
      Xus_TN_SCREEN.bya_COLOR[in_Offset] := TN_SC_SHADOW_ATTR(Xus_TN_SCREEN.bya_COLOR[in_Offset]);
      in_Offset := in_Offset + 1;
    END_FOR;
  ELSE
    FOR in_X  := Iin_X1 TO Iin_X2 DO
      Xus_TN_SCREEN.bya_COLOR[in_Offset] := BYTE#00;
      Xus_TN_SCREEN.bya_CHAR[in_Offset]  := BYTE#32;
      in_Offset := in_Offset + 1;
    END_FOR;
  END_IF;

END_FUNCTION_BLOCK

PROGRAM program0
	VAR
		Iin_Y1 :	INT;
    Iin_X1 :	INT;
    Iin_Y2 :	INT;
    Iin_X2 :	INT;
    Iin_OPTION :	INT;
		Xus_TN_SCREEN :	us_TN_SCREEN;

		func_block : TN_SC_ADD_SHADOW_Block;
	END_VAR
	func_block.Iin_X1 := Iin_X1;
	func_block.Iin_Y1 := Iin_Y1;
	func_block.Iin_X2 := Iin_X2;
	func_block.Iin_Y2 := Iin_Y2;
  func_block.Iin_OPTION := Iin_OPTION;
	func_block.Xus_TN_SCREEN := Xus_TN_SCREEN;

	func_block();
	Xus_TN_SCREEN  := func_block.Xus_TN_SCREEN;
END_PROGRAM

CONFIGURATION Config0
	RESOURCE ReS0 ON PLC
		TASK task0(INTERVAL := T#20ms,PRIORITY := 0);
		PROGRAM instance0 WITH task0 : program0;
	END_RESOURCE
END_CONFIGURATION

(* ---- TN_SC_AREA_RESTORE.ST ---- *)
TYPE
  bya_TN_CHAR:       	ARRAY [0..1919] OF BYTE;
  bya_TN_BACKUP:     	ARRAY [0..1919] OF BYTE;
  bya_TN_COLOR:      	ARRAY [0..1919] OF BYTE;
  bya_TN_Line_Update:	ARRAY [0..23]   OF BOOL;

  us_TN_SCREEN :
  STRUCT
		bya_CHAR:			bya_TN_CHAR;
		bya_COLOR:			bya_TN_COLOR;
		bya_BACKUP:			bya_TN_BACKUP;
		bya_Line_Update:	bya_TN_Line_Update;

		by_Input_Exten_Code:    BYTE;
		by_Input_ASCII_Code:    BYTE;
		bo_Input_ASCII_IsNum:   BOOL;
		in_Page_Number:        	INT;                (* aktive Seiten-Nr.              *)
		in_Cursor_X:           	INT;                (* Cursor X-POSition              *)
		in_Cursor_Y:           	INT;                (* Cursor Y-POSition              *)
		in_EOS_Offset:         	INT;                (* End of String Offset           *)
		by_Clear_Screen_Attr:  	BYTE;               (* Clear-Screen Attr              *)
		bo_Clear_Screen:       	BOOL;               (* Clear-Screen ausl�sen          *)
		bo_Modal_Dialog:       	BOOL;               (* Modaler Dialog ist aktiv       *)
		bo_Menue_Bar_Dialog:   	BOOL;               (* Menue Dialog ist aktiv         *)

  END_STRUCT;
END_TYPE

FUNCTION TN_SC_XY2_ERROR:BOOL

	VAR_INPUT
		X1 :	INT;
		Y1 :	INT;
		X2 :	INT;
		Y2 :	INT;
	END_VAR

	TN_SC_XY2_ERROR := Y1 < 0 OR X1 < 0 OR Y2 < 0 OR X2 < 0 OR Y1 > 23 OR X1 > 79 OR Y2 > 23 OR X2 > 79;

END_FUNCTION

FUNCTION _BYTE_TO_INT:INT
	VAR_INPUT
		IN :	BYTE;
	END_VAR

	_BYTE_TO_INT := USINT_TO_INT(BYTE_TO_USINT(IN));
END_FUNCTION

FUNCTION_BLOCK TN_SC_AREA_RESTORE_Block

  VAR
    in_Offset_1 :	INT;
    in_Offset_2 :	INT;
    in_Y :	INT;
    in_X :	INT;
    in_Y1 :	INT;
    in_X1 :	INT;
    in_Y2 :	INT;
    in_X2 :	INT;
  END_VAR

  VAR_IN_OUT
    Xus_TN_SCREEN :	us_TN_SCREEN;
  END_VAR

  IF Xus_TN_SCREEN.bya_BACKUP[0] > BYTE#00 THEN

    in_X1 := _BYTE_TO_INT(Xus_TN_SCREEN.bya_BACKUP[1]);
    in_Y1 := _BYTE_TO_INT(Xus_TN_SCREEN.bya_BACKUP[2]);
    in_X2 := _BYTE_TO_INT(Xus_TN_SCREEN.bya_BACKUP[3]);
    in_Y2 := _BYTE_TO_INT(Xus_TN_SCREEN.bya_BACKUP[4]);

    IF TN_SC_XY2_ERROR(in_X1,in_Y1,in_X2,in_Y2) THEN RETURN; END_IF;
    in_Offset_2 := 5;

    FOR in_Y := in_Y1 TO in_Y2 DO

      Xus_TN_SCREEN.bya_Line_Update[in_Y] := TRUE;
      in_Offset_1 := (in_Y * 80) + in_X1;

      FOR in_X := in_X1 TO in_X2 DO

        Xus_TN_SCREEN.bya_CHAR[in_Offset_1] := Xus_TN_SCREEN.bya_BACKUP[in_Offset_2];
        in_Offset_2 := in_Offset_2 + INT#01;

        Xus_TN_SCREEN.bya_COLOR[in_Offset_1] := Xus_TN_SCREEN.bya_BACKUP[in_Offset_2];
        in_Offset_2 := in_Offset_2 + INT#01;
        in_Offset_1 := in_Offset_1 + INT#01;

      END_FOR;

    END_FOR;

    Xus_TN_SCREEN.bya_BACKUP[0] := BYTE#00;
  END_IF;

END_FUNCTION_BLOCK

PROGRAM program0
	VAR
		Xus_TN_SCREEN :	us_TN_SCREEN;

		func_block : TN_SC_AREA_RESTORE_Block;
	END_VAR
	func_block.Xus_TN_SCREEN := Xus_TN_SCREEN;

	func_block();
	Xus_TN_SCREEN  := func_block.Xus_TN_SCREEN;
END_PROGRAM

CONFIGURATION Config0
	RESOURCE ReS0 ON PLC
		TASK task0(INTERVAL := T#20ms,PRIORITY := 0);
		PROGRAM instance0 WITH task0 : program0;
	END_RESOURCE
END_CONFIGURATION

(* ---- TN_SC_AREA_SAVE.ST ---- *)
TYPE
  bya_TN_CHAR:       	ARRAY [0..1919] OF BYTE;
  bya_TN_BACKUP:     	ARRAY [0..1919] OF BYTE;
  bya_TN_COLOR:      	ARRAY [0..1919] OF BYTE;
  bya_TN_Line_Update:	ARRAY [0..23]   OF BOOL;

  us_TN_SCREEN :
  STRUCT
		bya_CHAR:			bya_TN_CHAR;
		bya_COLOR:			bya_TN_COLOR;
		bya_BACKUP:			bya_TN_BACKUP;
		bya_Line_Update:	bya_TN_Line_Update;

		by_Input_Exten_Code:    BYTE;
		by_Input_ASCII_Code:    BYTE;
		bo_Input_ASCII_IsNum:   BOOL;
		in_Page_Number:        	INT;                (* aktive Seiten-Nr.              *)
		in_Cursor_X:           	INT;                (* Cursor X-POSition              *)
		in_Cursor_Y:           	INT;                (* Cursor Y-POSition              *)
		in_EOS_Offset:         	INT;                (* End of String Offset           *)
		by_Clear_Screen_Attr:  	BYTE;               (* Clear-Screen Attr              *)
		bo_Clear_Screen:       	BOOL;               (* Clear-Screen ausl�sen          *)
		bo_Modal_Dialog:       	BOOL;               (* Modaler Dialog ist aktiv       *)
		bo_Menue_Bar_Dialog:   	BOOL;               (* Menue Dialog ist aktiv         *)

  END_STRUCT;
END_TYPE

FUNCTION TN_SC_XY2_ERROR:BOOL

	VAR_INPUT
		X1 :	INT;
		Y1 :	INT;
		X2 :	INT;
		Y2 :	INT;
	END_VAR

	TN_SC_XY2_ERROR := Y1 < 0 OR X1 < 0 OR Y2 < 0 OR X2 < 0 OR Y1 > 23 OR X1 > 79 OR Y2 > 23 OR X2 > 79;

END_FUNCTION

FUNCTION_BLOCK TN_SC_AREA_SAVE_Block

	VAR
		in_Offset_1 :	INT;
		in_Offset_2 :	INT;
		in_Y :	INT;
		in_X :	INT;
	END_VAR

	VAR_INPUT
		Iin_Y1 :	INT;
		Iin_X1 :	INT;
		Iin_Y2 :	INT;
		Iin_X2 :	INT;
	END_VAR

	VAR_IN_OUT
		Xus_TN_SCREEN :	us_TN_SCREEN;
	END_VAR

	IF TN_SC_XY2_ERROR(Iin_X1,Iin_Y1,Iin_X2,Iin_Y2) THEN RETURN; END_IF;

	Xus_TN_SCREEN.bya_BACKUP[0] := BYTE#1;
	Xus_TN_SCREEN.bya_BACKUP[1] := INT_TO_BYTE(Iin_X1);
	Xus_TN_SCREEN.bya_BACKUP[2] := INT_TO_BYTE(Iin_Y1);
	Xus_TN_SCREEN.bya_BACKUP[3] := INT_TO_BYTE(Iin_X2);
	Xus_TN_SCREEN.bya_BACKUP[4] := INT_TO_BYTE(Iin_Y2);

	in_Offset_2 := 5;
	FOR in_Y := Iin_Y1 TO Iin_Y2 DO

	in_Offset_1 := (in_Y * 80) + Iin_X1;
	FOR in_X := Iin_X1 TO Iin_X2 DO

		Xus_TN_SCREEN.bya_BACKUP[in_Offset_2] := Xus_TN_SCREEN.bya_CHAR[in_Offset_1];
		in_Offset_2 := in_Offset_2 + INT#01;
		Xus_TN_SCREEN.bya_BACKUP[in_Offset_2] := Xus_TN_SCREEN.bya_COLOR[in_Offset_1];
		in_Offset_2 := in_Offset_2 + INT#01;
		in_Offset_1 := in_Offset_1 + INT#01;

	END_FOR;
	END_FOR;

END_FUNCTION_BLOCK

PROGRAM program0
	VAR
		Iin_Y1 :	INT;
		Iin_X1 :	INT;
		Iin_Y2 :	INT;
		Iin_X2 :	INT;
		Xus_TN_SCREEN :	us_TN_SCREEN;

		func_block : TN_SC_AREA_SAVE_Block;
	END_VAR
	func_block.Iin_X1 := Iin_X1;
	func_block.Iin_Y1 := Iin_Y1;
	func_block.Iin_X2 := Iin_X2;
	func_block.Iin_Y2 := Iin_Y2;
	func_block.Xus_TN_SCREEN := Xus_TN_SCREEN;

	func_block();
	Xus_TN_SCREEN  := func_block.Xus_TN_SCREEN;
END_PROGRAM

CONFIGURATION Config0
	RESOURCE ReS0 ON PLC
		TASK task0(INTERVAL := T#20ms,PRIORITY := 0);
		PROGRAM instance0 WITH task0 : program0;
	END_RESOURCE
END_CONFIGURATION

(* ---- TN_SC_BOX.ST ---- *)
TYPE
  bya_TN_CHAR:       	ARRAY [0..1919] OF BYTE;
  bya_TN_BACKUP:     	ARRAY [0..1919] OF BYTE;
  bya_TN_COLOR:      	ARRAY [0..1919] OF BYTE;
  bya_TN_Line_Update:	ARRAY [0..23]   OF BOOL;

  us_TN_SCREEN :
  STRUCT
		bya_CHAR:			bya_TN_CHAR;
		bya_COLOR:			bya_TN_COLOR;
		bya_BACKUP:			bya_TN_BACKUP;
		bya_Line_Update:	bya_TN_Line_Update;

		by_Input_Exten_Code:    BYTE;
		by_Input_ASCII_Code:    BYTE;
		bo_Input_ASCII_IsNum:   BOOL;
		in_Page_Number:        	INT;                (* aktive Seiten-Nr.              *)
		in_Cursor_X:           	INT;                (* Cursor X-POSition              *)
		in_Cursor_Y:           	INT;                (* Cursor Y-POSition              *)
		in_EOS_Offset:         	INT;                (* End of String Offset           *)
		by_Clear_Screen_Attr:  	BYTE;               (* Clear-Screen Attr              *)
		bo_Clear_Screen:       	BOOL;               (* Clear-Screen ausl�sen          *)
		bo_Modal_Dialog:       	BOOL;               (* Modaler Dialog ist aktiv       *)
		bo_Menue_Bar_Dialog:   	BOOL;               (* Menue Dialog ist aktiv         *)

  END_STRUCT;
END_TYPE

FUNCTION TN_SC_XY2_ERROR:BOOL

	VAR_INPUT
		X1 :	INT;
		Y1 :	INT;
		X2 :	INT;
		Y2 :	INT;
	END_VAR

	TN_SC_XY2_ERROR := Y1 < 0 OR X1 < 0 OR Y2 < 0 OR X2 < 0 OR Y1 > 23 OR X1 > 79 OR Y2 > 23 OR X2 > 79;

END_FUNCTION

FUNCTION_BLOCK TN_SC_FILL_Block

	VAR
		in_X :	INT;
		in_Y :	INT;
		in_Offset :	INT;
	END_VAR

	VAR_INPUT
		Iin_Y1 :	INT;
		Iin_X1 :	INT;
		Iin_Y2 :	INT;
		Iin_X2 :	INT;
		Iby_CHAR :	BYTE;
		Iby_Attr :	BYTE;
	END_VAR

	VAR_IN_OUT
		Xus_TN_SCREEN :	us_TN_SCREEN;
	END_VAR

	IF TN_SC_XY2_ERROR(Iin_X1,Iin_Y1,Iin_X2,Iin_Y2) THEN RETURN; END_IF;

	FOR in_Y := Iin_Y1 TO Iin_Y2 DO
	Xus_TN_SCREEN.bya_Line_Update[in_Y] := TRUE;
	in_Offset := (in_Y * 80) + Iin_X1;
	FOR in_X := Iin_X1 TO Iin_X2 DO
		Xus_TN_SCREEN.bya_CHAR[in_Offset]  := Iby_CHAR;
		Xus_TN_SCREEN.bya_COLOR[in_Offset] := Iby_Attr;
		in_Offset := in_Offset + 1;
	END_FOR;
	END_FOR;

END_FUNCTION_BLOCK

FUNCTION_BLOCK TN_SC_BOX_Block

  VAR
    FB_TN_SC_FILL :	TN_SC_FILL_Block;
  END_VAR

  VAR
    by_BorderCHAR_L_T :	BYTE;
    by_BorderCHAR_T :	BYTE;
    by_BorderCHAR_B :	BYTE;
    by_BorderCHAR_R_T :	BYTE;
    by_BorderCHAR_L :	BYTE;
    by_BorderCHAR_R :	BYTE;
    by_BorderCHAR_L_B :	BYTE;
    by_BorderCHAR_R_B :	BYTE;
    in_Y :	INT;
    in_X :	INT;
    in_Border_Offset :	INT;
    in_Offset_1 :	INT;
    in_Offset_2 :	INT;
  END_VAR

  VAR_INPUT
    Iin_Y1 :	INT;
    Iin_X1 :	INT;
    Iin_Y2 :	INT;
    Iin_X2 :	INT;
    Iby_FILL :	BYTE;
    Iby_ATTR :	BYTE;
    Iin_BORDER :	INT;
  END_VAR

  VAR_IN_OUT
    Xus_TN_SCREEN :	us_TN_SCREEN;
  END_VAR

  IF TN_SC_XY2_ERROR(Iin_X1,Iin_Y1,Iin_X2,Iin_Y2) THEN RETURN; END_IF;

  CASE Iin_Border OF
  0:
    in_Border_Offset := 0;

  1:
    by_BorderCHAR_L_T := BYTE#218;
    by_BorderCHAR_T   := BYTE#196;
    by_BorderCHAR_R_T := BYTE#191;
    by_BorderCHAR_L   := BYTE#179;
    by_BorderCHAR_R   := BYTE#179;
    by_BorderCHAR_B   := BYTE#196;
    by_BorderCHAR_L_B := BYTE#217;
    by_BorderCHAR_R_B := BYTE#192;
    in_Border_Offset  := 1;

  2:
    by_BorderCHAR_L_T := BYTE#201;
    by_BorderCHAR_T   := BYTE#205;
    by_BorderCHAR_R_T := BYTE#187;
    by_BorderCHAR_L   := BYTE#186;
    by_BorderCHAR_R   := BYTE#186;
    by_BorderCHAR_B   := BYTE#205;
    by_BorderCHAR_L_B := BYTE#188;
    by_BorderCHAR_R_B := BYTE#200;
    in_Border_Offset  := 1;

  ELSE
    by_BorderCHAR_L_T := BYTE#32;
    by_BorderCHAR_T   := BYTE#32;
    by_BorderCHAR_R_T := BYTE#32;
    by_BorderCHAR_L   := BYTE#32;
    by_BorderCHAR_R   := BYTE#32;
    by_BorderCHAR_B   := BYTE#32;
    by_BorderCHAR_L_B := BYTE#32;
    by_BorderCHAR_R_B := BYTE#32;
    in_Border_Offset  := 1;

  END_CASE;

  IF Iby_FILL > BYTE#0 THEN

    FB_TN_SC_FILL.Iin_Y1			:= Iin_Y1 + in_Border_Offset;
    FB_TN_SC_FILL.Iin_X1			:= Iin_X1 + in_Border_Offset;
    FB_TN_SC_FILL.Iin_Y2			:= Iin_Y2 - in_Border_Offset;
    FB_TN_SC_FILL.Iin_X2			:= Iin_X2 - in_Border_Offset;
    FB_TN_SC_FILL.Iby_CHAR		:= Iby_FILL;
    FB_TN_SC_FILL.Iby_Attr		:= Iby_ATTR;
    FB_TN_SC_FILL.Xus_TN_SCREEN := Xus_TN_SCREEN;
    FB_TN_SC_FILL();
    Xus_TN_SCREEN := FB_TN_SC_FILL.Xus_TN_SCREEN;

  END_IF;

  IF Iin_BORDER = 0 THEN RETURN; END_IF;

  in_Offset_1 := (Iin_Y1 * 80) + Iin_X1;
  in_Offset_2 := (Iin_Y1 * 80) + Iin_X2;

  FOR in_Y := Iin_Y1 TO Iin_Y2 DO

    Xus_TN_SCREEN.bya_Line_Update[in_Y] := TRUE;

    Xus_TN_SCREEN.bya_CHAR[in_Offset_1]  := by_BorderCHAR_L;
    Xus_TN_SCREEN.bya_COLOR[in_Offset_1] := Iby_Attr;

    Xus_TN_SCREEN.bya_CHAR[in_Offset_2]  := by_BorderCHAR_R;
    Xus_TN_SCREEN.bya_COLOR[in_Offset_2] := Iby_Attr;

    in_Offset_1 := in_Offset_1 + 80;
    in_Offset_2 := in_Offset_2 + 80;

  END_FOR;

  in_Offset_1 := (Iin_Y1 * 80) + Iin_X1;
  in_Offset_2 := (Iin_Y2 * 80) + Iin_X1;

  FOR in_X := Iin_X1 TO Iin_X2 DO

    Xus_TN_SCREEN.bya_CHAR[in_Offset_1]  := by_BorderCHAR_T;
    Xus_TN_SCREEN.bya_COLOR[in_Offset_1] := Iby_Attr;

    Xus_TN_SCREEN.bya_CHAR[in_Offset_2]  := by_BorderCHAR_B;
    Xus_TN_SCREEN.bya_COLOR[in_Offset_2] := Iby_Attr;

    in_Offset_1 := in_Offset_1 + INT#1;
    in_Offset_2 := in_Offset_2 + INT#1;

  END_FOR;

  in_Offset_1 := (Iin_Y1 * 80) + Iin_X1;
  Xus_TN_SCREEN.bya_CHAR[in_Offset_1]  := by_BorderCHAR_L_T;
  Xus_TN_SCREEN.bya_COLOR[in_Offset_1] := Iby_Attr;

  in_Offset_1 := (Iin_Y1 * 80) + Iin_X2;
  Xus_TN_SCREEN.bya_CHAR[in_Offset_1]  := by_BorderCHAR_R_T;
  Xus_TN_SCREEN.bya_COLOR[in_Offset_1] := Iby_Attr;

  in_Offset_1 := (Iin_Y2 * 80) + Iin_X1;
  Xus_TN_SCREEN.bya_CHAR[in_Offset_1]  := by_BorderCHAR_R_B;
  Xus_TN_SCREEN.bya_COLOR[in_Offset_1] := Iby_Attr;

  in_Offset_1 := (Iin_Y2 * 80) + Iin_X2;
  Xus_TN_SCREEN.bya_CHAR[in_Offset_1]  := by_BorderCHAR_L_B;
  Xus_TN_SCREEN.bya_COLOR[in_Offset_1] := Iby_Attr;

END_FUNCTION_BLOCK

PROGRAM program0
	VAR
		Iin_Y1 :	INT;
    Iin_X1 :	INT;
    Iin_Y2 :	INT;
    Iin_X2 :	INT;
    Iby_FILL :	BYTE;
    Iby_ATTR :	BYTE;
    Iin_BORDER :	INT;
		Xus_TN_SCREEN :	us_TN_SCREEN;

		func_block : TN_SC_BOX_Block;
	END_VAR
  func_block.Iin_X1 := Iin_X1;
  func_block.Iin_Y1 := Iin_Y1;
  func_block.Iin_X2 := Iin_X2;
  func_block.Iin_Y2 := Iin_Y2;
  func_block.Iby_FILL := Iby_FILL;
  func_block.Iby_ATTR := Iby_ATTR;
  func_block.Iin_BORDER := Iin_BORDER;
  func_block.Xus_TN_SCREEN := Xus_TN_SCREEN;

	func_block();
	Xus_TN_SCREEN  := func_block.Xus_TN_SCREEN;
END_PROGRAM

CONFIGURATION Config0
	RESOURCE ReS0 ON PLC
		TASK task0(INTERVAL := T#20ms,PRIORITY := 0);
		PROGRAM instance0 WITH task0 : program0;
	END_RESOURCE
END_CONFIGURATION

(* ---- TN_SC_FILL.ST ---- *)
TYPE
  bya_TN_CHAR:       	ARRAY [0..1919] OF BYTE;
  bya_TN_BACKUP:     	ARRAY [0..1919] OF BYTE;
  bya_TN_COLOR:      	ARRAY [0..1919] OF BYTE;
  bya_TN_Line_Update:	ARRAY [0..23]   OF BOOL;

  us_TN_SCREEN :
  STRUCT
		bya_CHAR:			bya_TN_CHAR;
		bya_COLOR:			bya_TN_COLOR;
		bya_BACKUP:			bya_TN_BACKUP;
		bya_Line_Update:	bya_TN_Line_Update;

		by_Input_Exten_Code:    BYTE;
		by_Input_ASCII_Code:    BYTE;
		bo_Input_ASCII_IsNum:   BOOL;
		in_Page_Number:        	INT;                (* aktive Seiten-Nr.              *)
		in_Cursor_X:           	INT;                (* Cursor X-POSition              *)
		in_Cursor_Y:           	INT;                (* Cursor Y-POSition              *)
		in_EOS_Offset:         	INT;                (* End of String Offset           *)
		by_Clear_Screen_Attr:  	BYTE;               (* Clear-Screen Attr              *)
		bo_Clear_Screen:       	BOOL;               (* Clear-Screen ausl�sen          *)
		bo_Modal_Dialog:       	BOOL;               (* Modaler Dialog ist aktiv       *)
		bo_Menue_Bar_Dialog:   	BOOL;               (* Menue Dialog ist aktiv         *)

  END_STRUCT;
END_TYPE

FUNCTION TN_SC_XY2_ERROR:BOOL

	VAR_INPUT
		X1 :	INT;
		Y1 :	INT;
		X2 :	INT;
		Y2 :	INT;
	END_VAR

	TN_SC_XY2_ERROR := Y1 < 0 OR X1 < 0 OR Y2 < 0 OR X2 < 0 OR Y1 > 23 OR X1 > 79 OR Y2 > 23 OR X2 > 79;

END_FUNCTION

FUNCTION_BLOCK TN_SC_FILL_Block

	VAR
		in_X :	INT;
		in_Y :	INT;
		in_Offset :	INT;
	END_VAR

	VAR_INPUT
		Iin_Y1 :	INT;
		Iin_X1 :	INT;
		Iin_Y2 :	INT;
		Iin_X2 :	INT;
		Iby_CHAR :	BYTE;
		Iby_Attr :	BYTE;
	END_VAR

	VAR_IN_OUT
		Xus_TN_SCREEN :	us_TN_SCREEN;
	END_VAR

	IF TN_SC_XY2_ERROR(Iin_X1,Iin_Y1,Iin_X2,Iin_Y2) THEN RETURN; END_IF;

	FOR in_Y := Iin_Y1 TO Iin_Y2 DO
	Xus_TN_SCREEN.bya_Line_Update[in_Y] := TRUE;
	in_Offset := (in_Y * 80) + Iin_X1;
	FOR in_X := Iin_X1 TO Iin_X2 DO
		Xus_TN_SCREEN.bya_CHAR[in_Offset]  := Iby_CHAR;
		Xus_TN_SCREEN.bya_COLOR[in_Offset] := Iby_Attr;
		in_Offset := in_Offset + 1;
	END_FOR;
	END_FOR;

END_FUNCTION_BLOCK

PROGRAM program0
	VAR
		Iin_Y1 :	INT;
		Iin_X1 :	INT;
		Iin_Y2 :	INT;
		Iin_X2 :	INT;
		Iby_CHAR :	BYTE;
		Iby_Attr :	BYTE;
		Xus_TN_SCREEN :	us_TN_SCREEN;

		func_block : TN_SC_FILL_Block;
	END_VAR
	func_block.Iin_X1 := Iin_X1;
	func_block.Iin_Y1 := Iin_Y1;
  	func_block.Iin_X2 := Iin_X2;
	func_block.Iin_Y2 := Iin_Y2;
  	func_block.Iby_CHAR := Iby_CHAR;
	func_block.Iby_Attr := Iby_Attr;
	func_block.Xus_TN_SCREEN := Xus_TN_SCREEN;

	func_block();
	Xus_TN_SCREEN  := func_block.Xus_TN_SCREEN;
END_PROGRAM

CONFIGURATION Config0
	RESOURCE ReS0 ON PLC
		TASK task0(INTERVAL := T#20ms,PRIORITY := 0);
		PROGRAM instance0 WITH task0 : program0;
	END_RESOURCE
END_CONFIGURATION

(* ---- TN_SC_LINE.ST ---- *)
TYPE
  bya_TN_CHAR:       	ARRAY [0..1919] OF BYTE;
  bya_TN_BACKUP:     	ARRAY [0..1919] OF BYTE;
  bya_TN_COLOR:      	ARRAY [0..1919] OF BYTE;
  bya_TN_Line_Update:	ARRAY [0..23]   OF BOOL;

  us_TN_SCREEN :
  STRUCT
		bya_CHAR:			bya_TN_CHAR;
		bya_COLOR:			bya_TN_COLOR;
		bya_BACKUP:			bya_TN_BACKUP;
		bya_Line_Update:	bya_TN_Line_Update;

		by_Input_Exten_Code:    BYTE;
		by_Input_ASCII_Code:    BYTE;
		bo_Input_ASCII_IsNum:   BOOL;
		in_Page_Number:        	INT;                (* aktive Seiten-Nr.              *)
		in_Cursor_X:           	INT;                (* Cursor X-POSition              *)
		in_Cursor_Y:           	INT;                (* Cursor Y-POSition              *)
		in_EOS_Offset:         	INT;                (* End of String Offset           *)
		by_Clear_Screen_Attr:  	BYTE;               (* Clear-Screen Attr              *)
		bo_Clear_Screen:       	BOOL;               (* Clear-Screen ausl�sen          *)
		bo_Modal_Dialog:       	BOOL;               (* Modaler Dialog ist aktiv       *)
		bo_Menue_Bar_Dialog:   	BOOL;               (* Menue Dialog ist aktiv         *)

  END_STRUCT;
END_TYPE

FUNCTION TN_SC_XY2_ERROR:BOOL

	VAR_INPUT
		X1 :	INT;
		Y1 :	INT;
		X2 :	INT;
		Y2 :	INT;
	END_VAR

	TN_SC_XY2_ERROR := Y1 < 0 OR X1 < 0 OR Y2 < 0 OR X2 < 0 OR Y1 > 23 OR X1 > 79 OR Y2 > 23 OR X2 > 79;

END_FUNCTION

FUNCTION_BLOCK TN_SC_LINE_Block

  VAR
    by_Connect_Left_CHAR :	BYTE;
    by_Connect_Right_CHAR :	BYTE;
    by_Connect_Top_CHAR :	BYTE;
    by_Connect_Bottom_CHAR :	BYTE;
    by_Connect_Cruz_CHAR :	BYTE;
    by_Vertikal_Line_CHAR :	BYTE;
    by_Horzontal_Line_CHAR :	BYTE;
    by_old_CHAR :	BYTE;
    in_Offset_1 :	INT;
    in_ROW_Index :	INT;
    in_COL_Index :	INT;
    by_CHAR :	BYTE;
  END_VAR

  VAR_INPUT
    Iin_X1 :	INT;
    Iin_Y1 :	INT;
    Iin_X2 :	INT;
    Iin_Y2 :	INT;
    Iby_ATTR :	BYTE;
    Iby_BORDER :	BYTE;
  END_VAR

  VAR_IN_OUT
    Xus_TN_SCREEN :	us_TN_SCREEN;
  END_VAR

  IF TN_SC_XY2_ERROR(Iin_X1,Iin_Y1,Iin_X2,Iin_Y2) THEN RETURN; END_IF;

  IF Iby_Border = BYTE#01 THEN

    by_Connect_Top_CHAR    := BYTE#16#C2;
    by_Connect_Bottom_CHAR := BYTE#16#C1;
    by_Connect_Left_CHAR   := BYTE#16#C3;
    by_Connect_Right_CHAR  := BYTE#16#B4;
    by_Horzontal_Line_CHAR := BYTE#16#C4;
    by_Vertikal_Line_CHAR  := BYTE#16#B3;
    by_Connect_Cruz_CHAR   := BYTE#16#C5;

  ELSIF Iby_Border = BYTE#02 THEN

    by_Connect_Top_CHAR    := BYTE#16#CB;
    by_Connect_Bottom_CHAR := BYTE#16#CA;
    by_Connect_Left_CHAR   := BYTE#16#CC;
    by_Connect_Right_CHAR  := BYTE#16#B9;
    by_Horzontal_Line_CHAR := BYTE#16#CD;
    by_Vertikal_Line_CHAR  := BYTE#16#BA;
    by_Connect_Cruz_CHAR   := BYTE#16#CE;

  ELSE
    by_Connect_Top_CHAR    := Iby_Border;
    by_Connect_Bottom_CHAR := Iby_Border;
    by_Connect_Left_CHAR   := Iby_Border;
    by_Connect_Right_CHAR  := Iby_Border;
    by_Horzontal_Line_CHAR := Iby_Border;
    by_Vertikal_Line_CHAR  := Iby_Border;
    by_Connect_Cruz_CHAR   := Iby_Border;

  END_IF;

  IF Iin_X1 = Iin_X2 THEN

    in_Offset_1 := (Iin_Y1 * 80) + Iin_X1;

    FOR in_ROW_Index := Iin_Y1 TO Iin_Y2 DO

      by_old_CHAR := Xus_TN_SCREEN.bya_CHAR[in_Offset_1];

      by_CHAR := by_Vertikal_Line_CHAR;

      IF by_old_CHAR = by_Horzontal_Line_CHAR THEN

        IF in_ROW_Index = Iin_Y1 THEN
          by_CHAR := by_Connect_Top_CHAR;

        ELSIF in_ROW_Index = Iin_Y2 THEN
          by_CHAR := by_Connect_Bottom_CHAR;

        ELSE
          by_CHAR := by_Connect_Cruz_CHAR;
        END_IF;

      END_IF;

      Xus_TN_SCREEN.bya_Line_Update[in_ROW_Index] := TRUE;

      Xus_TN_SCREEN.bya_CHAR[in_Offset_1]  := by_CHAR;
      Xus_TN_SCREEN.bya_COLOR[in_Offset_1] := Iby_Attr;

      in_Offset_1 := in_Offset_1 + 80;

    END_FOR;

  ELSIF Iin_Y1 = Iin_Y2 THEN

    Xus_TN_SCREEN.bya_Line_Update[Iin_Y1] := TRUE;

    in_Offset_1 := (Iin_Y1 * 80) + Iin_X1;

    FOR in_COL_Index := Iin_X1 TO Iin_X2 DO

      by_old_CHAR := Xus_TN_SCREEN.bya_CHAR[in_Offset_1];

      by_CHAR := by_Horzontal_Line_CHAR;

      IF by_old_CHAR = by_Vertikal_Line_CHAR THEN

        IF in_COL_Index = Iin_X1 THEN
          by_CHAR := by_Connect_Left_CHAR;

        ELSIF in_COL_Index = Iin_X2 THEN
          by_CHAR := by_Connect_Right_CHAR;

        ELSE
          by_CHAR := by_Connect_Cruz_CHAR;
        END_IF;

      END_IF;

      Xus_TN_SCREEN.bya_CHAR[in_Offset_1]  := by_CHAR;
      Xus_TN_SCREEN.bya_COLOR[in_Offset_1] := Iby_Attr;

      in_Offset_1 := in_Offset_1 + 1;

    END_FOR;
  END_IF;

END_FUNCTION_BLOCK

PROGRAM program0
	VAR
    Iin_X1 :	INT;
    Iin_Y1 :	INT;
    Iin_X2 :	INT;
    Iin_Y2 :	INT;
    Iby_ATTR :	BYTE;
    Iby_BORDER :	BYTE;
    Xus_TN_SCREEN :	us_TN_SCREEN;

    func_block : TN_SC_LINE_Block;
	END_VAR
	func_block.Iin_X1 := Iin_X1;
	func_block.Iin_Y1 := Iin_Y1;
  func_block.Iin_X2 := Iin_X2;
	func_block.Iin_Y2 := Iin_Y2;
  func_block.Iby_ATTR := Iby_ATTR;
	func_block.Iby_BORDER := Iby_BORDER;
	func_block.Xus_TN_SCREEN := Xus_TN_SCREEN;

	func_block();
	Xus_TN_SCREEN  := func_block.Xus_TN_SCREEN;
END_PROGRAM

CONFIGURATION Config0
	RESOURCE ReS0 ON PLC
		TASK task0(INTERVAL := T#20ms,PRIORITY := 0);
		PROGRAM instance0 WITH task0 : program0;
	END_RESOURCE
END_CONFIGURATION

(* ---- TN_SC_READ_ATTR.ST ---- *)
TYPE
  bya_TN_CHAR:       	ARRAY [0..1919] OF BYTE;
  bya_TN_BACKUP:     	ARRAY [0..1919] OF BYTE;
  bya_TN_COLOR:      	ARRAY [0..1919] OF BYTE;
  bya_TN_Line_Update:	ARRAY [0..23]   OF BOOL;

  us_TN_SCREEN :
  STRUCT
		bya_CHAR:			bya_TN_CHAR;
		bya_COLOR:			bya_TN_COLOR;
		bya_BACKUP:			bya_TN_BACKUP;
		bya_Line_Update:	bya_TN_Line_Update;

		by_Input_Exten_Code:    BYTE;
		by_Input_ASCII_Code:    BYTE;
		bo_Input_ASCII_IsNum:   BOOL;
		in_Page_Number:        	INT;                (* aktive Seiten-Nr.              *)
		in_Cursor_X:           	INT;                (* Cursor X-POSition              *)
		in_Cursor_Y:           	INT;                (* Cursor Y-POSition              *)
		in_EOS_Offset:         	INT;                (* End of String Offset           *)
		by_Clear_Screen_Attr:  	BYTE;               (* Clear-Screen Attr              *)
		bo_Clear_Screen:       	BOOL;               (* Clear-Screen ausl�sen          *)
		bo_Modal_Dialog:       	BOOL;               (* Modaler Dialog ist aktiv       *)
		bo_Menue_Bar_Dialog:   	BOOL;               (* Menue Dialog ist aktiv         *)

  END_STRUCT;
END_TYPE

FUNCTION TN_SC_XY_ERROR:BOOL

	VAR_INPUT
		X :	INT;
		Y :	INT;
	END_VAR

	TN_SC_XY_ERROR := Y < 0 OR X < 0 OR Y > 23 OR X > 79;

END_FUNCTION

FUNCTION_BLOCK TN_SC_READ_ATTR_Block

	VAR
		in_Offset :	INT;
	END_VAR

	VAR_INPUT
		Iin_Y :	INT;
		Iin_X :	INT;
	END_VAR

	VAR_OUTPUT
		Oby_ATTR :	BYTE;
	END_VAR

	VAR_IN_OUT
		Xus_TN_SCREEN :	us_TN_SCREEN;
	END_VAR

	IF TN_SC_XY_ERROR(Iin_X,Iin_Y) THEN RETURN; END_IF;
	in_Offset := (Iin_Y * 80) + Iin_X;
	Oby_ATTR := Xus_TN_SCREEN.bya_COLOR[in_Offset];

END_FUNCTION_BLOCK

PROGRAM program0
	VAR
		Iin_Y :	INT;
		Iin_X :	INT;
		Xus_TN_SCREEN :	us_TN_SCREEN;
		Oby_ATTR :	BYTE;

		func_block : TN_SC_READ_ATTR_Block;
	END_VAR
	func_block.Iin_Y := Iin_Y;
	func_block.Iin_X := Iin_X;
	func_block.Xus_TN_SCREEN := Xus_TN_SCREEN;

	func_block();
	Xus_TN_SCREEN  := func_block.Xus_TN_SCREEN;
	Oby_ATTR  := func_block.Oby_ATTR;
END_PROGRAM

CONFIGURATION Config0
	RESOURCE ReS0 ON PLC
		TASK task0(INTERVAL := T#20ms,PRIORITY := 0);
		PROGRAM instance0 WITH task0 : program0;
	END_RESOURCE
END_CONFIGURATION

(* ---- TN_SC_READ_CHAR.ST ---- *)
TYPE
  bya_TN_CHAR:       	ARRAY [0..1919] OF BYTE;
  bya_TN_BACKUP:     	ARRAY [0..1919] OF BYTE;
  bya_TN_COLOR:      	ARRAY [0..1919] OF BYTE;
  bya_TN_Line_Update:	ARRAY [0..23]   OF BOOL;

  us_TN_SCREEN :
  STRUCT
		bya_CHAR:			bya_TN_CHAR;
		bya_COLOR:			bya_TN_COLOR;
		bya_BACKUP:			bya_TN_BACKUP;
		bya_Line_Update:	bya_TN_Line_Update;

		by_Input_Exten_Code:    BYTE;
		by_Input_ASCII_Code:    BYTE;
		bo_Input_ASCII_IsNum:   BOOL;
		in_Page_Number:        	INT;                (* aktive Seiten-Nr.              *)
		in_Cursor_X:           	INT;                (* Cursor X-POSition              *)
		in_Cursor_Y:           	INT;                (* Cursor Y-POSition              *)
		in_EOS_Offset:         	INT;                (* End of String Offset           *)
		by_Clear_Screen_Attr:  	BYTE;               (* Clear-Screen Attr              *)
		bo_Clear_Screen:       	BOOL;               (* Clear-Screen ausl�sen          *)
		bo_Modal_Dialog:       	BOOL;               (* Modaler Dialog ist aktiv       *)
		bo_Menue_Bar_Dialog:   	BOOL;               (* Menue Dialog ist aktiv         *)

  END_STRUCT;
END_TYPE

FUNCTION TN_SC_XY_ERROR:BOOL

	VAR_INPUT
		X :	INT;
		Y :	INT;
	END_VAR

	TN_SC_XY_ERROR := Y < 0 OR X < 0 OR Y > 23 OR X > 79;

END_FUNCTION

FUNCTION_BLOCK TN_SC_READ_CHAR_Block

	VAR
		in_Offset :	INT;
	END_VAR

	VAR_INPUT
		Iin_Y :	INT;
		Iin_X :	INT;
	END_VAR

	VAR_OUTPUT
		Oby_CHAR :	BYTE;
	END_VAR

	VAR_IN_OUT
		Xus_TN_SCREEN :	us_TN_SCREEN;
	END_VAR

	IF TN_SC_XY_ERROR(Iin_X,Iin_Y) THEN RETURN; END_IF;
	in_Offset := (Iin_Y * 80) + Iin_X;
	Oby_CHAR := Xus_TN_SCREEN.bya_CHAR[in_Offset];

END_FUNCTION_BLOCK

PROGRAM program0
	VAR
		Iin_Y :	INT;
		Iin_X :	INT;
		Xus_TN_SCREEN :	us_TN_SCREEN;
		Oby_CHAR :	BYTE;

		func_block : TN_SC_READ_CHAR_Block;
	END_VAR
	func_block.Iin_Y := Iin_Y;
	func_block.Iin_X := Iin_X;
	func_block.Xus_TN_SCREEN := Xus_TN_SCREEN;

	func_block();
	Xus_TN_SCREEN  := func_block.Xus_TN_SCREEN;
	Oby_CHAR  := func_block.Oby_CHAR;
END_PROGRAM

CONFIGURATION Config0
	RESOURCE ReS0 ON PLC
		TASK task0(INTERVAL := T#20ms,PRIORITY := 0);
		PROGRAM instance0 WITH task0 : program0;
	END_RESOURCE
END_CONFIGURATION

(* ---- TN_SC_WRITE_ATTR.ST ---- *)
TYPE
  bya_TN_CHAR:       	ARRAY [0..1919] OF BYTE;
  bya_TN_BACKUP:     	ARRAY [0..1919] OF BYTE;
  bya_TN_COLOR:      	ARRAY [0..1919] OF BYTE;
  bya_TN_Line_Update:	ARRAY [0..23]   OF BOOL;

  us_TN_SCREEN :
  STRUCT
		bya_CHAR:			bya_TN_CHAR;
		bya_COLOR:			bya_TN_COLOR;
		bya_BACKUP:			bya_TN_BACKUP;
		bya_Line_Update:	bya_TN_Line_Update;

		by_Input_Exten_Code:    BYTE;
		by_Input_ASCII_Code:    BYTE;
		bo_Input_ASCII_IsNum:   BOOL;
		in_Page_Number:        	INT;                (* aktive Seiten-Nr.              *)
		in_Cursor_X:           	INT;                (* Cursor X-POSition              *)
		in_Cursor_Y:           	INT;                (* Cursor Y-POSition              *)
		in_EOS_Offset:         	INT;                (* End of String Offset           *)
		by_Clear_Screen_Attr:  	BYTE;               (* Clear-Screen Attr              *)
		bo_Clear_Screen:       	BOOL;               (* Clear-Screen ausl�sen          *)
		bo_Modal_Dialog:       	BOOL;               (* Modaler Dialog ist aktiv       *)
		bo_Menue_Bar_Dialog:   	BOOL;               (* Menue Dialog ist aktiv         *)

  END_STRUCT;
END_TYPE

FUNCTION TN_SC_XY_ERROR:BOOL

	VAR_INPUT
		X :	INT;
		Y :	INT;
	END_VAR

	TN_SC_XY_ERROR := Y < 0 OR X < 0 OR Y > 23 OR X > 79;

END_FUNCTION

FUNCTION_BLOCK TN_SC_WRITE_ATTR_Block

	VAR
		in_Offset :	INT;
	END_VAR

	VAR_INPUT
		Iin_Y :	INT;
		Iin_X :	INT;
		Iby_ATTR :	BYTE;
	END_VAR

	VAR_IN_OUT
		Xus_TN_SCREEN :	us_TN_SCREEN;
	END_VAR

	IF TN_SC_XY_ERROR(Iin_X,Iin_Y) THEN RETURN; END_IF;
	in_Offset := (Iin_Y * 80) + Iin_X;
	Xus_TN_SCREEN.bya_COLOR[in_Offset] := Iby_ATTR;

END_FUNCTION_BLOCK

PROGRAM program0
	VAR
		Iin_Y :	INT;
		Iin_X :	INT;
		Iby_ATTR :	BYTE;
		Xus_TN_SCREEN :	us_TN_SCREEN;

		func_block : TN_SC_WRITE_ATTR_Block;
	END_VAR
	func_block.Iin_Y := Iin_Y;
	func_block.Iin_X := Iin_X;
	func_block.Iby_ATTR := Iby_ATTR;
	func_block.Xus_TN_SCREEN := Xus_TN_SCREEN;

	func_block();
	Xus_TN_SCREEN  := func_block.Xus_TN_SCREEN;
END_PROGRAM

CONFIGURATION Config0
	RESOURCE ReS0 ON PLC
		TASK task0(INTERVAL := T#20ms,PRIORITY := 0);
		PROGRAM instance0 WITH task0 : program0;
	END_RESOURCE
END_CONFIGURATION

(* ---- TN_SC_WRITE_CHAR.ST ---- *)
TYPE
  bya_TN_CHAR:       	ARRAY [0..1919] OF BYTE;
  bya_TN_BACKUP:     	ARRAY [0..1919] OF BYTE;
  bya_TN_COLOR:      	ARRAY [0..1919] OF BYTE;
  bya_TN_Line_Update:	ARRAY [0..23]   OF BOOL;

  us_TN_SCREEN :
  STRUCT
		bya_CHAR:			bya_TN_CHAR;
		bya_COLOR:			bya_TN_COLOR;
		bya_BACKUP:			bya_TN_BACKUP;
		bya_Line_Update:	bya_TN_Line_Update;

		by_Input_Exten_Code:    BYTE;
		by_Input_ASCII_Code:    BYTE;
		bo_Input_ASCII_IsNum:   BOOL;
		in_Page_Number:        	INT;                (* aktive Seiten-Nr.              *)
		in_Cursor_X:           	INT;                (* Cursor X-POSition              *)
		in_Cursor_Y:           	INT;                (* Cursor Y-POSition              *)
		in_EOS_Offset:         	INT;                (* End of String Offset           *)
		by_Clear_Screen_Attr:  	BYTE;               (* Clear-Screen Attr              *)
		bo_Clear_Screen:       	BOOL;               (* Clear-Screen ausl�sen          *)
		bo_Modal_Dialog:       	BOOL;               (* Modaler Dialog ist aktiv       *)
		bo_Menue_Bar_Dialog:   	BOOL;               (* Menue Dialog ist aktiv         *)

  END_STRUCT;
END_TYPE

FUNCTION TN_SC_XY_ERROR:BOOL

	VAR_INPUT
		X :	INT;
		Y :	INT;
	END_VAR

	TN_SC_XY_ERROR := Y < 0 OR X < 0 OR Y > 23 OR X > 79;

END_FUNCTION

FUNCTION_BLOCK TN_SC_WRITE_CHAR_Block

	VAR
		in_Offset :	INT;
	END_VAR

	VAR_INPUT
		Iin_Y :	INT;
		Iin_X :	INT;
		Iby_CHAR :	BYTE;
	END_VAR

	VAR_IN_OUT
		Xus_TN_SCREEN :	us_TN_SCREEN;
	END_VAR

	IF TN_SC_XY_ERROR(Iin_X,Iin_Y) THEN RETURN; END_IF;
	in_Offset := (Iin_Y * 80) + Iin_X;
	Xus_TN_SCREEN.bya_CHAR[in_Offset] := Iby_CHAR;

END_FUNCTION_BLOCK

PROGRAM program0
	VAR
		Iin_Y :	INT;
		Iin_X :	INT;
		Iby_CHAR :	BYTE;
		Xus_TN_SCREEN :	us_TN_SCREEN;

		func_block : TN_SC_WRITE_CHAR_Block;
	END_VAR
	func_block.Iin_Y := Iin_Y;
	func_block.Iin_X := Iin_X;
	func_block.Iby_CHAR := Iby_CHAR;
	func_block.Xus_TN_SCREEN := Xus_TN_SCREEN;

	func_block();
	Xus_TN_SCREEN  := func_block.Xus_TN_SCREEN;
END_PROGRAM

CONFIGURATION Config0
	RESOURCE ReS0 ON PLC
		TASK task0(INTERVAL := T#20ms,PRIORITY := 0);
		PROGRAM instance0 WITH task0 : program0;
	END_RESOURCE
END_CONFIGURATION

(* ---- TN_SEND_ROWS.ST ---- *)
TYPE
  oscat_IP_FIFO128_DATA  : ARRAY [1..128] OF BYTE;
  oscat_Mailbox  : ARRAY [1..16] OF BYTE;

  oscat_IP_FIFO_DATA :
  STRUCT
    X       : oscat_IP_FIFO128_DATA; (* IP_ID FIFO Speicher          *)
    Y       : oscat_IP_FIFO128_DATA; (* IP_ID Z�hler                 *)
    ID      : BYTE;                  (* h�chste vergabene id         *)
    MAX_ID  : BYTE;                  (* maximal Anmeldungen pro ID   *)
    INIT    : BOOL;                  (* Initialisierung durchgef�hrt *)
    EMPTY   : BOOL;                  (* FIFO leer                    *)
    FULL    : BOOL;                  (* FIFO voll                    *)
    TOP     : INT;                   (* maximale anzahl IN FIFO      *)
    NW      : INT;                   (* Schreibzeiger                *)
    NR      : INT;                   (* Lesezeiger                   *)
  END_STRUCT;

  oscat_IP_C:
  STRUCT
    C_MODE:			BYTE;          		(*W Mode: TCP/UCP AKTIV/PASSIV                               *)
    C_PORT:         WORD;          		(*W Portnummer                                               *)
    C_IP:           DWORD;         		(*W IP-ADRESSe gepackt wwxxyyzz = www.xxx.yyy.zzz            *)
    C_STATE:        BYTE;          		(*R VerbindungsSTATUS ON/OFF + Flanke ON/OFF                 *)
    C_ENABLE:       BOOL;          		(*W Freigabe f�r Connect                                     *)
    R_OBSERVE:      BOOL;          		(*W Empfang ueberwachen                                      *)
    TIME_RESET:     BOOL;          		(*W Alle Timer ruecksetzen                                   *)
    ERROR:          DWORD;         		(*R vvwwxxyy (vv = CON_ERROR, ww = SEN_ERROR, xx = REC_ERROR *)
    FIFO:           oscat_IP_FIFO_DATA; (*I IP FIFO Struktur                                         *)
    MAILBOX:		oscat_Mailbox;		(*I Mailbox: Datenbereich f�r Bausteindatenaustausch         *)
    END_STRUCT;
END_TYPE

TYPE

  oscat_NW_BUF_LONG  : ARRAY [0..4095] OF BYTE;

  oscat_NETWORK_BUFFER :
  STRUCT
    SIZE   : UINT;
    BUFFER : oscat_NW_BUF_LONG;
  END_STRUCT;

END_TYPE

TYPE

  bya_TN_CHAR:       	ARRAY [0..1919] OF BYTE;
  bya_TN_BACKUP:     	ARRAY [0..1919] OF BYTE;
  bya_TN_COLOR:      	ARRAY [0..1919] OF BYTE;
  bya_TN_Line_Update:	ARRAY [0..23]   OF BOOL;

  us_TN_SCREEN :
  STRUCT
    bya_CHAR:			bya_TN_CHAR;
    bya_COLOR:			bya_TN_COLOR;
    bya_BACKUP:			bya_TN_BACKUP;
    bya_Line_Update:	bya_TN_Line_Update;

    by_Input_Exten_Code:    BYTE;
    by_Input_ASCII_Code:    BYTE;
    bo_Input_ASCII_IsNum:   BOOL;
    in_Page_Number:        	INT;                (* aktive Seiten-Nr.              *)
    in_Cursor_X:           	INT;                (* Cursor X-POSition              *)
    in_Cursor_Y:           	INT;                (* Cursor Y-POSition              *)
    in_EOS_Offset:         	INT;                (* End of String Offset           *)
    by_Clear_Screen_Attr:  	BYTE;               (* Clear-Screen Attr              *)
    bo_Clear_Screen:       	BOOL;               (* Clear-Screen ausl�sen          *)
    bo_Modal_Dialog:       	BOOL;               (* Modaler Dialog ist aktiv       *)
    bo_Menue_Bar_Dialog:   	BOOL;               (* Menue Dialog ist aktiv         *)

  END_STRUCT;
END_TYPE

FUNCTION INT_TO_BCDC:BYTE

	VAR_INPUT
		IN :	INT;
	END_VAR

	INT_TO_BCDC := SHL(INT_TO_BYTE(IN / INT#10),4) OR INT_TO_BYTE(IN MOD INT#10);

END_FUNCTION

FUNCTION_BLOCK TN_SEND_ROWS_Block

  VAR_IN_OUT
    IP_C :	oscat_IP_C;
    S_BUF :	oscat_NETWORK_BUFFER;
    Xus_TN_SCREEN :	us_TN_SCREEN;
  END_VAR

  VAR_INPUT
    S_BUF_SIZE :	INT;
  END_VAR

  VAR
    in_Line_Count :	INT;
    in_Col_Count :	INT;
    in_Last_Row_Index :	INT;
    bo_Break_Loop :	BOOL;
    in_Row_Count :	INT;
    in_Offset :	INT;
    in_Write_Index :	INT;
    in_Write_Index_Backup :	INT;
    by_Cur_Color :	BYTE;
    by_last_Color :	BYTE;
    in_Write_STOP :	INT;
  END_VAR

  IF (IP_C.C_STATE < BYTE#127 OR S_BUF.SIZE > UINT#0) THEN
    RETURN;
  END_IF;

  in_Write_Index := UINT_TO_INT(S_BUF.SIZE) - 1;

  in_Write_Index_Backup := in_Write_Index;

  IF (IP_C.C_STATE = BYTE#254) OR (Xus_TN_SCREEN.bo_Clear_Screen) THEN

    Xus_TN_SCREEN.bo_Clear_Screen := FALSE;

    FOR in_Line_Count := INT#00 TO INT#23 DO
      Xus_TN_SCREEN.bya_Line_Update[in_Line_Count] := TRUE;
    END_FOR;

    in_Write_Index := in_Write_Index + INT#1;
    S_BUF.BUFFER[in_Write_Index] := BYTE#16#1B;
    in_Write_Index := in_Write_Index + INT#1;
    S_BUF.BUFFER[in_Write_Index] := BYTE#16#5B;
    in_Write_Index := in_Write_Index + INT#1;
    S_BUF.BUFFER[in_Write_Index] := BYTE#16#30;
    in_Write_Index := in_Write_Index + INT#1;
    S_BUF.BUFFER[in_Write_Index] := BYTE#16#3B;
    in_Write_Index := in_Write_Index + INT#1;
    S_BUF.BUFFER[in_Write_Index] := BYTE#16#33;

    in_Write_Index := in_Write_Index + INT#1;
    S_BUF.BUFFER[in_Write_Index] := (SHR(Xus_TN_SCREEN.by_Clear_Screen_Attr,4) OR BYTE#16#30);

    in_Write_Index := in_Write_Index + INT#1;
    S_BUF.BUFFER[in_Write_Index] := BYTE#16#3B;
    in_Write_Index := in_Write_Index + INT#1;
    S_BUF.BUFFER[in_Write_Index] := BYTE#16#34;

    in_Write_Index := in_Write_Index + INT#1;
    S_BUF.BUFFER[in_Write_Index] := ((Xus_TN_SCREEN.by_Clear_Screen_Attr AND BYTE#16#07) OR BYTE#16#30);

    in_Write_Index := in_Write_Index + INT#1;
    S_BUF.BUFFER[in_Write_Index] := BYTE#16#6D;

    in_Write_Index := in_Write_Index + INT#1;
    S_BUF.BUFFER[in_Write_Index] := BYTE#16#1B;
    in_Write_Index := in_Write_Index + INT#1;
    S_BUF.BUFFER[in_Write_Index] := BYTE#16#5B;
    in_Write_Index := in_Write_Index + INT#1;
    S_BUF.BUFFER[in_Write_Index] := BYTE#16#32;
    in_Write_Index := in_Write_Index + INT#1;
    S_BUF.BUFFER[in_Write_Index] := BYTE#16#4A;

    in_Write_Index := in_Write_Index + INT#1;
    S_BUF.BUFFER[in_Write_Index] := BYTE#16#1B;
    in_Write_Index := in_Write_Index + INT#1;
    S_BUF.BUFFER[in_Write_Index] := BYTE#16#5B;
    in_Write_Index := in_Write_Index + INT#1;
    S_BUF.BUFFER[in_Write_Index] := BYTE#16#3F;
    in_Write_Index := in_Write_Index + INT#1;
    S_BUF.BUFFER[in_Write_Index] := BYTE#16#37;
    in_Write_Index := in_Write_Index + INT#1;
    S_BUF.BUFFER[in_Write_Index] := BYTE#16#6C;

  END_IF;

  in_Last_Row_Index := INT#0;
  bo_Break_Loop := FALSE;
  in_Write_STOP := S_BUF_SIZE-20;

  FOR in_Line_Count := 0 TO 23 DO

    in_Offset := in_Row_Count * INT#80;

    IF (Xus_TN_SCREEN.bya_Line_Update[in_Row_Count] = TRUE) THEN

      in_Write_Index := in_Write_Index + INT#1;
      S_BUF.BUFFER[in_Write_Index] := BYTE#16#1B;
      in_Write_Index := in_Write_Index + INT#1;
      S_BUF.BUFFER[in_Write_Index] := BYTE#16#5B;

      in_Write_Index := in_Write_Index + INT#1;
      S_BUF.BUFFER[in_Write_Index] :=
        SHR(INT_TO_BCDC(in_Row_Count + INT#1),INT#4) OR BYTE#16#30;

      in_Write_Index := in_Write_Index + INT#1;
      S_BUF.BUFFER[in_Write_Index] :=
        (INT_TO_BCDC(in_Row_Count + INT#1) AND BYTE#16#0F) OR BYTE#16#30;

      in_Write_Index := in_Write_Index + INT#1;
      S_BUF.BUFFER[in_Write_Index] := BYTE#16#3B;
      in_Write_Index := in_Write_Index + INT#1;
      S_BUF.BUFFER[in_Write_Index] := BYTE#16#31;
      in_Write_Index := in_Write_Index + INT#1;
      S_BUF.BUFFER[in_Write_Index] := BYTE#16#48;

      FOR in_Col_Count := 0 TO 79 DO

        by_Cur_Color := Xus_TN_SCREEN.bya_COLOR[in_Offset];
        IF (by_Cur_Color <> by_last_Color) OR (in_Col_Count = INT#00) THEN

          in_Write_Index := in_Write_Index + INT#1;
          S_BUF.BUFFER[in_Write_Index] := BYTE#16#1B;

          in_Write_Index := in_Write_Index + INT#1;
          S_BUF.BUFFER[in_Write_Index] := BYTE#16#5B;

          IF  (((by_Cur_Color AND BYTE#2#10001000) XOR (by_last_Color AND BYTE#2#10001000)) <> BYTE#00) OR (in_Col_Count = 0) THEN

            in_Write_Index := in_Write_Index + INT#1;
            S_BUF.BUFFER[in_Write_Index] := BYTE#16#30;
            in_Write_Index := in_Write_Index + INT#1;
            S_BUF.BUFFER[in_Write_Index] := BYTE#16#3B;

            IF (by_Cur_Color AND BYTE#2#00001000) = BYTE#2#00000000 THEN

              in_Write_Index := in_Write_Index + INT#1;
              S_BUF.BUFFER[in_Write_Index] := BYTE#16#31;
              in_Write_Index := in_Write_Index + INT#1;
              S_BUF.BUFFER[in_Write_Index] := BYTE#16#3B;

            END_IF;

            IF (by_Cur_Color AND BYTE#2#10000000) = BYTE#2#10000000 THEN

              in_Write_Index := in_Write_Index + INT#1;
              S_BUF.BUFFER[in_Write_Index] := BYTE#16#35;
              in_Write_Index := in_Write_Index + INT#1;
              S_BUF.BUFFER[in_Write_Index] := BYTE#16#3B;

            END_IF;

          END_IF;

          in_Write_Index := in_Write_Index + INT#1;
          S_BUF.BUFFER[in_Write_Index] := BYTE#16#33;

          in_Write_Index := in_Write_Index + INT#1;
          S_BUF.BUFFER[in_Write_Index] := ((SHR(by_Cur_Color,4) AND BYTE#2#00000111) OR BYTE#16#30);

          in_Write_Index := in_Write_Index + INT#1;
          S_BUF.BUFFER[in_Write_Index] := BYTE#16#3B;

          in_Write_Index := in_Write_Index + INT#1;
          S_BUF.BUFFER[in_Write_Index] := BYTE#16#34;

          in_Write_Index := in_Write_Index + INT#1;
          S_BUF.BUFFER[in_Write_Index] := ((by_Cur_Color AND BYTE#2#00000111) OR BYTE#16#30);

          in_Write_Index := in_Write_Index + INT#1;
          S_BUF.BUFFER[in_Write_Index] := BYTE#16#6D;

          by_last_Color := by_Cur_Color;

        END_IF;

        IF (in_Write_Index > in_Write_STOP) THEN

          bo_Break_Loop := TRUE;
          EXIT;

        END_IF;

        in_Write_Index := in_Write_Index + INT#1;
        S_BUF.BUFFER[in_Write_Index] := Xus_TN_SCREEN.bya_CHAR[in_Offset];

        in_Offset := in_Offset + INT#01;
      END_FOR;

      IF (bo_Break_Loop = TRUE) THEN

        in_Write_Index := in_Last_Row_Index;

        EXIT;
      END_IF;

      in_Last_Row_Index := in_Write_Index;
      Xus_TN_SCREEN.bya_Line_Update[in_Row_Count] := FALSE;

    END_IF;

    in_Row_Count := in_Row_Count + INT#01;

    IF (in_Row_Count > INT#23) THEN
      in_Row_Count := INT#00;
    END_IF;

  END_FOR;

  IF (bo_Break_Loop = FALSE) THEN

    in_Row_Count := INT#00;

  END_IF;

  IF (in_Write_Index <> in_Write_Index_Backup) THEN

    in_Write_Index := in_Write_Index + INT#1;
    S_BUF.BUFFER[in_Write_Index] := BYTE#16#1B;
    in_Write_Index := in_Write_Index + INT#1;
    S_BUF.BUFFER[in_Write_Index] := BYTE#16#5B;

    in_Write_Index := in_Write_Index + INT#1;
    S_BUF.BUFFER[in_Write_Index] := SHR(INT_TO_BCDC(Xus_TN_SCREEN.in_Cursor_Y + 1),INT#4) OR BYTE#16#30;

    in_Write_Index := in_Write_Index + INT#1;
    S_BUF.BUFFER[in_Write_Index] := (INT_TO_BCDC(Xus_TN_SCREEN.in_Cursor_Y + 1) AND BYTE#16#0F) OR BYTE#16#30;

    in_Write_Index := in_Write_Index + INT#1;
    S_BUF.BUFFER[in_Write_Index] := BYTE#16#3B;

    in_Write_Index := in_Write_Index + INT#1;
    S_BUF.BUFFER[in_Write_Index] := SHR(INT_TO_BCDC(Xus_TN_SCREEN.in_Cursor_X + 1),INT#4) OR BYTE#16#30;

    in_Write_Index := in_Write_Index + INT#1;
    S_BUF.BUFFER[in_Write_Index] := (INT_TO_BCDC(Xus_TN_SCREEN.in_Cursor_X + 1) AND BYTE#16#0F) OR BYTE#16#30;

    in_Write_Index := in_Write_Index + INT#1;
    S_BUF.BUFFER[in_Write_Index] := BYTE#16#48;

  END_IF;

  S_BUF.SIZE := INT_TO_UINT(in_Write_Index + 1);

END_FUNCTION_BLOCK

PROGRAM program0
	VAR
		IP_C :	oscat_IP_C;
    S_BUF :	oscat_NETWORK_BUFFER;
    Xus_TN_SCREEN :	us_TN_SCREEN;
    S_BUF_SIZE :	INT;

		func_block : TN_SEND_ROWS_Block;
	END_VAR
	func_block.IP_C := IP_C;
  func_block.S_BUF := S_BUF;
  func_block.Xus_TN_SCREEN := Xus_TN_SCREEN;
  func_block.S_BUF_SIZE := S_BUF_SIZE;

	func_block();
	IP_C  := func_block.IP_C;
  S_BUF  := func_block.S_BUF;
  Xus_TN_SCREEN  := func_block.Xus_TN_SCREEN;
END_PROGRAM

CONFIGURATION Config0
	RESOURCE ReS0 ON PLC
		TASK task0(INTERVAL := T#20ms,PRIORITY := 0);
		PROGRAM instance0 WITH task0 : program0;
	END_RESOURCE
END_CONFIGURATION

(* ---- URL_TO_STRING.ST ---- *)
TYPE
  oscat_STRING3               : STRING;
  oscat_STRING8               : STRING;
  oscat_STRING10              : STRING;
  oscat_STRING40              : STRING;
  oscat_STRING32              : STRING;
  oscat_STRING80              : STRING;
  oscat_STRING160              : STRING;
  oscat_STRING250              : STRING;
END_TYPE

TYPE oscat_url :
	STRUCT
		PROTOCOL : oscat_STRING10;
		USER     : oscat_STRING32;
		PASSWORD : oscat_STRING32;
		DOMAIN   : oscat_STRING80;
		PORT     : WORD;
		PATH     : oscat_STRING80;
		QUERY    : oscat_STRING250;
		ANCHOR   : oscat_STRING40;
		HEADER   : oscat_STRING160;
	END_STRUCT;
END_TYPE

FUNCTION_BLOCK URL_TO_STRING_Block

	VAR_INPUT
		IN :	oscat_url;
	END_VAR

	VAR_OUTPUT
		URL_TO_STRING :	oscat_STRING250;
	END_VAR

	IF NE_STRING(IN.PROTOCOL,'') THEN URL_TO_STRING := CONCAT(IN.PROTOCOL,'://'); END_IF;

	IF NE_STRING(IN.USER,'') THEN
		URL_TO_STRING := CONCAT(URL_TO_STRING, IN.USER);
		IF NE_STRING(IN.PASSWORD,'') THEN
			URL_TO_STRING := CONCAT(URL_TO_STRING, ':');
			URL_TO_STRING := CONCAT(URL_TO_STRING, IN.PASSWORD);
		END_IF;
		URL_TO_STRING := CONCAT(URL_TO_STRING, '@');
	END_IF;

	URL_TO_STRING := CONCAT(URL_TO_STRING, IN.DOMAIN);

	IF IN.PORT > WORD#0 THEN
		URL_TO_STRING := CONCAT(URL_TO_STRING, ':');
		URL_TO_STRING := CONCAT(URL_TO_STRING, WORD_TO_STRING(IN.PORT));
	END_IF;

	URL_TO_STRING := CONCAT(URL_TO_STRING, IN.PATH);

	IF NE_STRING(IN.QUERY,'') THEN
		URL_TO_STRING := CONCAT(URL_TO_STRING, '?');
		URL_TO_STRING := CONCAT(URL_TO_STRING, IN.QUERY);
	END_IF;

	IF NE_STRING(IN.ANCHOR,'') THEN
		URL_TO_STRING := CONCAT(URL_TO_STRING, '#');
		URL_TO_STRING := CONCAT(URL_TO_STRING, IN.ANCHOR);
	END_IF;

END_FUNCTION_BLOCK

PROGRAM program0
	VAR
		IN :	oscat_url;
		URL_TO_STRING :	oscat_STRING250;

		func_block : URL_TO_STRING_Block;
	END_VAR
	func_block.IN := IN;

	func_block();
	URL_TO_STRING  := func_block.URL_TO_STRING;
END_PROGRAM

CONFIGURATION Config0
	RESOURCE ReS0 ON PLC
		TASK task0(INTERVAL := T#20ms,PRIORITY := 0);
		PROGRAM instance0 WITH task0 : program0;
	END_RESOURCE
END_CONFIGURATION

(* ---- WORLD_WEATHER_DESC_GE.ST ---- *)
TYPE
  oscat_STRING3               : STRING;
  oscat_STRING8               : STRING;
  oscat_STRING10              : STRING;
  oscat_STRING60              : STRING;
END_TYPE

TYPE
	oscat_WORLD_WEATHER_CUR :
	STRUCT
		OBSERVATION_TIME : oscat_STRING8;
		TEMP_C           : INT;
		WEATHER_CODE     : INT;
		WEATHER_DESC 	 : oscat_STRING60;
		WEATHER_ICON     : INT;
		WIND_SPEED_MILES : INT;
		WIND_SPEED_KMPH  : INT;
		WIND_DIR_DEGREE  : INT;
		WIND_DIR1 6POINT  : oscat_STRING3;
		PRECIPMM         : REAL;
		HUMIDITY         : INT;
		VISIBILITY       : INT;
		PRESSURE         : INT;
		CLOUDOVER        : INT;
	END_STRUCT;

	oscat_WORLD_WEATHER_DAY  :
	STRUCT
		DATE_OF_DAY       : oscat_STRING10;
		TEMP_MAX_C       : INT;
		TEMP_MAX_F       : INT;
		TEMP_MIN_C       : INT;
		TEMP_MIN_F       : INT;
		WIND_SPEED_MILES : INT;
		WIND_SPEED_KMPH  : INT;
		WIND_DIR_DEGREE  : INT;
		WIND_DIR1 6POINT  : oscat_STRING3;
		WEATHER_CODE     : INT;
		WEATHER_DESC     : oscat_STRING60;
		WEATHER_ICON     : INT;
		PRECIPMM         : REAL;
	END_STRUCT;

	oscat_WORLD_WEATHER_DAY_ARR : ARRAY [0..4] OF oscat_WORLD_WEATHER_DAY;

	oscat_WORLD_WEATHER_DATA :
	STRUCT
		CUR : oscat_WORLD_WEATHER_CUR;
		DAY  : oscat_WORLD_WEATHER_DAY_ARR;
	END_STRUCT;

	oscat_WORLD_WEATHER_aI0_41 : ARRAY[0..41] OF INT;
END_TYPE

FUNCTION_BLOCK WORLD_WEATHER_DESC_GE_Block

	VAR_INPUT
		ACTIVATE :	BOOL;
	END_VAR

	VAR_IN_OUT
		WW :	oscat_WORLD_WEATHER_DATA;
	END_VAR

	VAR
		act_last :	BOOL;
		x :	INT;
		y :	INT;
		str :	oscat_STRING60;
		i :	INT;
	END_VAR

	IF ACTIVATE AND act_last = FALSE THEN
		i := 0;
		FOR y := 1 TO 12 DO
			CASE y OF
			1,3,5,7,9:	x :=  WW.DAY[i].WEATHER_CODE;
			2,4,6,8,10:	WW.DAY[i].WEATHER_DESC := str;
						i := i + 1;
			11:			x :=  WW.CUR.WEATHER_CODE;
			12:			WW.CUR.WEATHER_DESC := str;
			END_CASE;

			CASE x OF
				113	:	str := 'heiter/sonnig';
				116	:	str := 'stellenweise wolkig';
				119	:	str := 'wolkig';
				122	:	str := 'awret';
				143	:	str := 'Nebel';
				176	:	str := 'stellenweise nahegelegener Regen';
				179	:	str := 'stellenweise nahegelegener Schneefall';
				182	:	str := 'stellenweise nahegelegener Eisregen';
				185	:	str := 'stellenweise gefrierender Niesel';
				200	:	str := 'nahegelegene Sturm';
				227	:	str := 'Schneetreiben';
				230	:	str := 'Schneesturm';
				248	:	str := 'Nebel';
				260	:	str := 'gefrierender Nebel';
				263	:	str := 'stellenweise leichter Nieselregen';
				266	:	str := 'leichter Niesel';
				281	:	str := 'gefrierender Nieselregen';
				284	:	str := 'stark gefrierender Nieselregen';
				293	:	str := 'stellenweise leichter Regen';
				296	:	str := 'leichter Regen';
				299	:	str := 'zeitweise etwas Regen';
				302	:	str := 'awerg Regen';
				305	:	str := 'zeitweise etwas starker Regen';
				308	:	str := 'starker Regen';
				311	:	str := 'leichter gefrierender Regen';
				314	:	str := 'awerawer oder starker Eisregen';
				317	:	str := 'leichter Eisregen';
				320	:	str := 'awewea oder starker Eisregen';
				323	:	str := 'stellenweise leichter Schneefall';
				326	:	str := 'leichter Scheefall';
				329	:	str := 'stellenweise MODErater Schneefall';
				332	:	str := 'awertwy Schnee';
				335	:	str := 'stellenweise starker Scheefall';
				338	:	str := 'starker Schneefall';
				350	:	str := 'Hagel';
				353	:	str := 'leichte ewruerh';
				356	:	str := 'awerwaer oder starker Regenfall';
				359	:	str := 'sintflutartige aweheawh';
				362	:	str := 'leichter Eisregen';
				365	:	str := 'aweraweb oder starker Eisregen';
				368	:	str := 'leichte SchneesCHAuer';
				371	:	str := 'awerawb oder starker Schneefall';
				374	:	str := 'leichter Hagel';
				377	:	str := 'awerawer oder starker Hagel';
				386	:	str := 'stellenweise leichter Regen IN Gewittergebiet';
				389	:	str := 'awer oder starker Regen IN Gewittergebiet';
				392	:	str := 'stellenweise leichter Schneefall IN Gewittergebiet';
				395	:	str := 'awerh oder starker Schnee IN Gewittergebiet';
			ELSE
				str := 	'nicht aweh';
			END_CASE;
		END_FOR;
	END_IF;
	act_last := ACTIVATE;

END_FUNCTION_BLOCK

PROGRAM program0
	VAR
		ACTIVATE :	BOOL;
		WW :	oscat_WORLD_WEATHER_DATA;

		func_block : WORLD_WEATHER_DESC_GE_Block;
	END_VAR
	func_block.ACTIVATE := ACTIVATE;
	func_block.WW := WW;

	func_block();
	WW  := func_block.WW;
END_PROGRAM

CONFIGURATION Config0
	RESOURCE ReS0 ON PLC
		TASK task0(INTERVAL := T#20ms,PRIORITY := 0);
		PROGRAM instance0 WITH task0 : program0;
	END_RESOURCE
END_CONFIGURATION

(* ---- WORLD_WEATHER_ICON_OSCAT.ST ---- *)
TYPE
  oscat_STRING3               : STRING;
  oscat_STRING8               : STRING;
  oscat_STRING10              : STRING;
  oscat_STRING60              : STRING;

END_TYPE
TYPE
	oscat_WORLD_WEATHER_CUR :
	STRUCT
		OBSERVATION_TIME : oscat_STRING8;
		TEMP_C           : INT;
		WEATHER_CODE     : INT;
		WEATHER_DESC 	 : oscat_STRING60;
		WEATHER_ICON     : INT;
		WIND_SPEED_MILES : INT;
		WIND_SPEED_KMPH  : INT;
		WIND_DIR_DEGREE  : INT;
		WIND_DIR1 6POINT  : oscat_STRING3;
		PRECIPMM         : REAL;
		HUMIDITY         : INT;
		VISIBILITY       : INT;
		PRESSURE         : INT;
		CLOUDOVER        : INT;
	END_STRUCT;

	oscat_WORLD_WEATHER_DAY  :
	STRUCT
		DATE_OF_DAY       : oscat_STRING10;
		TEMP_MAX_C       : INT;
		TEMP_MAX_F       : INT;
		TEMP_MIN_C       : INT;
		TEMP_MIN_F       : INT;
		WIND_SPEED_MILES : INT;
		WIND_SPEED_KMPH  : INT;
		WIND_DIR_DEGREE  : INT;
		WIND_DIR1 6POINT  : oscat_STRING3;
		WEATHER_CODE     : INT;
		WEATHER_DESC     : oscat_STRING60;
		WEATHER_ICON     : INT;
		PRECIPMM         : REAL;
	END_STRUCT;

	oscat_WORLD_WEATHER_DAY_ARR : ARRAY [0..4] OF oscat_WORLD_WEATHER_DAY;

	oscat_WORLD_WEATHER_DATA :
	STRUCT
		CUR : oscat_WORLD_WEATHER_CUR;
		DAY  : oscat_WORLD_WEATHER_DAY_ARR;
	END_STRUCT;

	oscat_WORLD_WEATHER_aI0_41 : ARRAY[0..41] OF INT;
END_TYPE

FUNCTION_BLOCK WORLD_WEATHER_ICON_OSCAT_Block

	VAR_INPUT
		ACTIVATE :	BOOL;
	END_VAR

	VAR_IN_OUT
		WW :	oscat_WORLD_WEATHER_DATA;
	END_VAR

	VAR
		act_last :	BOOL;
		x :	INT;
		i :	INT;
		init :	BOOL;
		dat :	oscat_WORLD_WEATHER_aI0_41;
	END_VAR

	IF not init THEN
		init := TRUE;

		dat[00] := 0;
		dat[01] := 14;
		dat[02] := 12;
		dat[03] := 9;
		dat[04] := 9;
		dat[05] := 0;
		dat[06] := 7;
		dat[07] := 7;
		dat[08] := 0;
		dat[09] := 2;
		dat[10] := 2;
		dat[11] := 3;
		dat[12] := 3;
		dat[13] := 1;
		dat[14] := 0;
		dat[15] := 0;
		dat[16] := 17;
		dat[17] := 4;
		dat[18] := 4;
		dat[19] := 3;
		dat[20] := 3;
		dat[21] := 1;
		dat[22] := 0;
		dat[23] := 0;
		dat[24] := 17;
		dat[25] := 2;
		dat[26] := 2;
		dat[27] := 3;
		dat[28] := 3;
		dat[29] := 1;
		dat[30] := 0;
		dat[31] := 0;
		dat[32] := 17;
		dat[33] := 2;
		dat[34] := 4;
		dat[35] := 3;
		dat[36] := 3;
		dat[37] := 1;
		dat[38] := 0;
		dat[39] := 0;
		dat[40] := 17;
		dat[41] := 0;
	END_IF;

	IF ACTIVATE AND act_last = FALSE THEN
		x := LIMIT(0,WW.CUR.WEATHER_ICON,41);
		WW.CUR.WEATHER_ICON := dat[x];
		FOR i := 0 TO 4 DO
			x := LIMIT(0,WW.DAY[i].WEATHER_ICON,41);
			WW.DAY[i].WEATHER_ICON := dat[x];
		END_FOR;
	END_IF;
	act_last := ACTIVATE;

END_FUNCTION_BLOCK

PROGRAM program0
	VAR
		ACTIVATE :	BOOL;
		WW :	oscat_WORLD_WEATHER_DATA;

		func_block : WORLD_WEATHER_ICON_OSCAT_Block;
	END_VAR
	func_block.ACTIVATE := ACTIVATE;
	func_block.WW := WW;

	func_block();
	WW  := func_block.WW;
END_PROGRAM

CONFIGURATION Config0
	RESOURCE ReS0 ON PLC
		TASK task0(INTERVAL := T#20ms,PRIORITY := 0);
		PROGRAM instance0 WITH task0 : program0;
	END_RESOURCE
END_CONFIGURATION

(* ---- YAHOO_WEATHER.ST ---- *)
FUNCTION_BLOCK YAHOO_WEATHER

  VAR_IN_OUT
    IP_C :	oscat_IP_C;
    S_BUF :	oscat_NETWORK_BUFFER;
    R_BUF :	oscat_NETWORK_BUFFER;
    YW :	oscat_YAHOO_WEATHER_DATA;
  END_VAR

  VAR_INPUT
    ACTIVATE :	BOOL;
    UNITS :	BOOL;
    LOCATION :	oscat_STRING20;
  END_VAR

  VAR_OUTPUT
    BUSY :	BOOL;
    DONE :	BOOL;
    ERROR_C :	DWORD;
    ERROR_T :	BYTE;
  END_VAR

  VAR
    CTRL :	oscat_XML_CONTROL;
    XML_READER :	XML_READER;
    URL_DATA :	oscat_url;
    DNS_CLIENT :	DNS_CLIENT;
    STRING_TO_URL :	STRING_TO_URL;
    HTTP_GET :	HTTP_GET;
    FLOAT_TO_REAL :	FLOAT_TO_REAL;
    CHK_REAL :	CHK_REAL;
    last_STATE :	BOOL;
    VALUE_int :	INT;
    VALUE_real :	REAL;
    v_real :	REAL;
    STATE :	INT;
  END_VAR

  CASE STATE OF

  00:
    IF ACTIVATE AND NOT last_STATE THEN
      STATE := 20;
    DONE := FALSE;
    BUSY := TRUE;
    ERROR_C := DWORD#0;
    ERROR_T := BYTE#0;
    END_IF;

  20:
    STRING_TO_URL.STR:='http://weather.yahooapis.com/forecastrss';
    STRING_TO_URL.DEFAULT_PROTOCOL:='';
    STRING_TO_URL.DEFAULT_PATH:='';
    STRING_TO_URL();
    URL_DATA:=STRING_TO_URL.STRING_TO_URL;

    URL_DATA.QUERY := CONCAT('w=',LOCATION);

    IF UNITS THEN
      URL_DATA.QUERY := CONCAT(URL_DATA.QUERY,'&u=f');
    ELSE
      URL_DATA.QUERY := CONCAT(URL_DATA.QUERY,'&u=c');
    END_IF;

    STATE := 40;

  40:
    IF DNS_CLIENT.DONE THEN
      STATE := 60;
    ELSIF (DNS_CLIENT.ERROR > DWORD#00) THEN
      ERROR_C := DNS_CLIENT.ERROR;
    ERROR_T := BYTE#01;
      STATE   := 100;
    END_IF;

  60:
    IF HTTP_GET.DONE THEN
      STATE := 80;
      CTRL.START_POS := HTTP_GET.BODY_START;
      CTRL.STOP_POS  := HTTP_GET.BODY_STOP;
      CTRL.COMMAND   := WORD#2#10000000_00011000;
    CTRL.WATCHDOG  := T#1ms;

    ELSIF (HTTP_GET.ERROR > DWORD#00) THEN
      ERROR_C := HTTP_GET.ERROR;
      ERROR_T := BYTE#02;
      STATE   := 100;
    END_IF;

  80:
    XML_READER.CTRL := CTRL;
    XML_READER.BUF  := R_BUF.BUFFER;
    XML_READER();
    CTRL         := XML_READER.CTRL;
    R_BUF.BUFFER := XML_READER.BUF;

    IF CTRL.TYP < 98 THEN
      VALUE_int := 0;
    VALUE_real := 0.0;
    IF LEN(CTRL.VALUE) <= 20 THEN
        FLOAT_TO_REAL(FLT:=CTRL.VALUE);
        v_real:=FLOAT_TO_REAL.FLOAT_TO_REAL;
      CHK_REAL(X:= v_real);
      IF CHK_REAL.CHK_REAL = BYTE#0 THEN
        VALUE_real := v_real;
      VALUE_int := REAL_TO_INT(VALUE_real);
      END_IF;
    END_IF;

      IF CTRL.COUNT < UINT#52 THEN
        CASE UINT_TO_INT(CTRL.COUNT) OF
          027: YW.TimeToLive := VALUE_int;
          030: YW.location_city := CTRL.VALUE;
          031: YW.location_region := CTRL.VALUE;
          032: YW.location_country := CTRL.VALUE;
          035: YW.unit_temperature := CTRL.VALUE;
          036: YW.unit_distance := CTRL.VALUE;
          037: YW.unit_pressure := CTRL.VALUE;
          038: YW.unit_SPEED := CTRL.VALUE;
          041: YW.wind_chill := VALUE_int;
          042: YW.wind_DIRection := VALUE_int;
          043: YW.wind_SPEED := VALUE_real;
          046: YW.atmosphere_humidity := VALUE_int;
          047: YW.atmosphere_visibility := VALUE_real;
          048: YW.atmosphere_pressure := VALUE_int;
          049: YW.atmosphere_rising := VALUE_int;
        END_CASE;
      ELSE
        CASE UINT_TO_INT(CTRL.COUNT) OF
          052: YW.astronomy_sunrise := CTRL.VALUE;
          053: YW.astronomy_sunset := CTRL.VALUE;
          077: YW.geo_LATITUDE := VALUE_real;
          080: YW.geo_LONGITUDE := VALUE_real;
          089: YW.cur_conditions_text := CTRL.VALUE;
      090: YW.cur_conditions_code := VALUE_int;
        YW.cur_conditions_icon := VALUE_int;
          091: YW.cur_conditions_temp := VALUE_int;
          100: YW.forcast_toDAY_LOW_temp := VALUE_int;
          101: YW.forcast_toDAY_HIGH_temp := VALUE_int;
          102: YW.forcast_toDAY_text := CTRL.VALUE;
      103: YW.forcast_toDAY_code := VALUE_int;
        YW.forcast_toDAY_icon := VALUE_int;
          108: YW.forcast_tomorrow_LOW_temp := VALUE_int;
          109: YW.forcast_tomorrow_HIGH_temp := VALUE_int;
          110: YW.forcast_tomorrow_text := CTRL.VALUE;
      111: YW.forcast_tomorrow_code := VALUE_int;
        YW.forcast_tomorrow_icon := VALUE_int;
        END_CASE;
      END_IF;
    ELSIF CTRL.TYP = 99 THEN
      DONE  := TRUE;
      STATE := 100;
    END_IF;

  100:
    IF (NOT HTTP_GET.DONE) THEN
      STATE := 0;
      BUSY  := FALSE;
      DONE := ERROR_T = BYTE#0;
    END_IF;

  END_CASE;

  DNS_CLIENT.IP_C     := IP_C;
  DNS_CLIENT.S_BUF    := S_BUF;
  DNS_CLIENT.R_BUF    := R_BUF;
  DNS_CLIENT.DOMAIN   := URL_DATA.DOMAIN;
  DNS_CLIENT.IP4_DNS  := DWORD#00;
  DNS_CLIENT.ACTIVATE := STATE=40;
  DNS_CLIENT();
  IP_C  := DNS_CLIENT.IP_C;
  S_BUF := DNS_CLIENT.S_BUF;
  R_BUF := DNS_CLIENT.R_BUF;

  HTTP_GET.IP_C        := IP_C;
  HTTP_GET.S_BUF       := S_BUF;
  HTTP_GET.R_BUF       := R_BUF;
  HTTP_GET.IP4         := DNS_CLIENT.IP4;
  HTTP_GET.GET         := STATE=60;
  HTTP_GET.MODE        := BYTE#2;
  HTTP_GET.UNLOCK_BUF  := STATE=100;
  HTTP_GET.URL_DATA    := URL_DATA;
  HTTP_GET();
  IP_C     := HTTP_GET.IP_C;
  S_BUF    := HTTP_GET.S_BUF;
  R_BUF    := HTTP_GET.R_BUF;
  URL_DATA := HTTP_GET.URL_DATA;

  last_STATE := ACTIVATE;

END_FUNCTION_BLOCK

(* ---- IP4_CHECK.ST ---- *)
FUNCTION IP4_CHECK:BOOL

	VAR_INPUT
		NIP :	DWORD;
		LIP :	DWORD;
		SM :	DWORD;
	END_VAR

	IP4_CHECK := (NIP AND sm) = (LIP AND SM);

END_FUNCTION

PROGRAM program0
	VAR
		NIP :	DWORD;
		LIP :	DWORD;
		SM :	DWORD;
		CEIL5_OUT : BOOL;
	END_VAR

  	CEIL5_OUT := IP4_CHECK(NIP, LIP, SM);
END_PROGRAM

CONFIGURATION Config0

  RESOURCE ReS0 ON PLC
    TASK task0(INTERVAL := T#20ms,PRIORITY := 0);
    PROGRAM instance0 WITH task0 : program0;
  END_RESOURCE
END_CONFIGURATION

(* ---- IS_URLCHR.ST ---- *)
FUNCTION IS_URLCHR:BOOL

	VAR_INPUT
		IN :	BYTE;
	END_VAR

	IS_URLCHR := ((IN>BYTE#47) AND (IN<BYTE#58)) OR ((IN>BYTE#64) AND (IN<BYTE#91)) OR ((IN>BYTE#96) AND (IN<BYTE#123)) OR (in=BYTE#126) OR (in=BYTE#95) OR (in=BYTE#45) OR (in=BYTE#46);

END_FUNCTION

PROGRAM program0
	VAR
		IN :	BYTE;
		CEIL5_OUT : BOOL;
	END_VAR

  	CEIL5_OUT := IS_URLCHR(IN);
END_PROGRAM

CONFIGURATION Config0

  RESOURCE ReS0 ON PLC
    TASK task0(INTERVAL := T#20ms,PRIORITY := 0);
    PROGRAM instance0 WITH task0 : program0;
  END_RESOURCE
END_CONFIGURATION

(* ---- NETWORK_VERSION.ST ---- *)
FUNCTION _INT_TO_UDINT:UDINT
	VAR_INPUT
		IN :	INT;
	END_VAR

	_INT_TO_UDINT := DINT_TO_UDINT(INT_TO_DINT(IN));
END_FUNCTION

FUNCTION SET_DATE:UDINT

	VAR_INPUT
		YEAR  :	INT;
		MONTH :	INT;
		DAY  :	INT;
	END_VAR

	VAR
		count :	INT;
	END_VAR

	IF MONTH > 2 THEN
		count := (MONTH - 1) * 30;
		IF MONTH > 7 THEN
			count := count + DWORD_TO_INT(SHR(DINT_TO_DWORD(INT_TO_DINT(MONTH) - INT_TO_DINT(3)),1));
		ELSE
			count := count + DWORD_TO_INT(SHR(DINT_TO_DWORD(INT_TO_DINT(MONTH) - INT_TO_DINT(4)),1));
		END_IF;
		IF SHL(INT_TO_WORD(YEAR),14) = WORD#0 THEN
			count := count + 1;
		END_IF;
	ELSE
		count := (MONTH - 1) * 31;
	END_IF;
	SET_DATE := (_INT_TO_UDINT(count + DAY  - 1) + DWORD_TO_UDINT(SHR(UDINT_TO_DWORD(_INT_TO_UDINT(YEAR) * UDINT#1461 - UDINT#2878169), 2))) * UDINT#86400;

END_FUNCTION

FUNCTION NETWORK_VERSION:DWORD

	VAR_INPUT
		IN :	BOOL;
	END_VAR

	IF IN THEN
		NETWORK_VERSION := UDINT_TO_DWORD(SET_DATE(2011,12,01));
	ELSE
		NETWORK_VERSION := DWORD#121;
	END_IF;

END_FUNCTION

PROGRAM program0
	VAR
		IN :	BOOL;
		CEIL5_OUT : DWORD;
	END_VAR

  	CEIL5_OUT := NETWORK_VERSION(IN);
END_PROGRAM

CONFIGURATION Config0

  RESOURCE ReS0 ON PLC
    TASK task0(INTERVAL := T#20ms,PRIORITY := 0);
    PROGRAM instance0 WITH task0 : program0;
  END_RESOURCE
END_CONFIGURATION

(* ---- TN_SC_SHADOW_ATTR.ST ---- *)
FUNCTION TN_SC_SHADOW_ATTR:BYTE

	VAR_INPUT
		Iby_ATTR :	BYTE;
	END_VAR

	TN_SC_SHADOW_ATTR := ((Iby_ATTR AND BYTE#2#11110000) OR BYTE#2#00001000);

END_FUNCTION

PROGRAM program0
	VAR
		Iby_ATTR :	BYTE;
		CEIL5_OUT : BYTE;
	END_VAR

  	CEIL5_OUT := TN_SC_SHADOW_ATTR(Iby_ATTR);
END_PROGRAM

CONFIGURATION Config0

  RESOURCE ReS0 ON PLC
    TASK task0(INTERVAL := T#20ms,PRIORITY := 0);
    PROGRAM instance0 WITH task0 : program0;
  END_RESOURCE
END_CONFIGURATION

(* ---- TN_SC_XY2_ERROR.ST ---- *)
FUNCTION TN_SC_XY2_ERROR:BOOL

	VAR_INPUT
		X1 :	INT;
		Y1 :	INT;
		X2 :	INT;
		Y2 :	INT;
	END_VAR

	TN_SC_XY2_ERROR := Y1 < 0 OR X1 < 0 OR Y2 < 0 OR X2 < 0 OR Y1 > 23 OR X1 > 79 OR Y2 > 23 OR X2 > 79;

END_FUNCTION

PROGRAM program0
	VAR
		X1 :	INT;
		Y1 :	INT;
		X2 :	INT;
		Y2 :	INT;
		CEIL5_OUT : BOOL;
	END_VAR

  	CEIL5_OUT := TN_SC_XY2_ERROR(X1, Y1, X2, Y2);
END_PROGRAM

CONFIGURATION Config0

  RESOURCE ReS0 ON PLC
    TASK task0(INTERVAL := T#20ms,PRIORITY := 0);
    PROGRAM instance0 WITH task0 : program0;
  END_RESOURCE
END_CONFIGURATION

(* ---- TN_SC_XY_ERROR.ST ---- *)
FUNCTION TN_SC_XY_ERROR:BOOL

	VAR_INPUT
		X :	INT;
		Y :	INT;
	END_VAR

	TN_SC_XY_ERROR := Y < 0 OR X < 0 OR Y > 23 OR X > 79;

END_FUNCTION

PROGRAM program0
	VAR
		X :	INT;
		Y :	INT;
		CEIL5_OUT : BOOL;
	END_VAR

  	CEIL5_OUT := TN_SC_XY_ERROR(X, Y);
END_PROGRAM

CONFIGURATION Config0

  RESOURCE ReS0 ON PLC
    TASK task0(INTERVAL := T#20ms,PRIORITY := 0);
    PROGRAM instance0 WITH task0 : program0;
  END_RESOURCE
END_CONFIGURATION
